(* CODESYS project XPlanarApplication206.library
   Version: 2.0.6
   Title: XPlanarApplication
   DefaultNamespace: XPlanarApplication
   Placeholder: XPlanarApplication
   Company: Beckhoff Automation LLC

Project tree, tasks and I/O mapping:
  libraries: Tc2_Math, * (Beckhoff Automation GmbH); Tc2_Standard, * (Beckhoff Automation GmbH); Tc2_System, * (Beckhoff Automation GmbH); Tc2_Utilities, * (Beckhoff Automation GmbH); Tc3_EventLogger, * (Beckhoff Automation GmbH); Tc3_Mc3PlanarMotion, * (Beckhoff Automation GmbH); Tc3_Module, * (Beckhoff Automation GmbH); Tc3_Physics, * (Beckhoff Automation GmbH); Tc3_XPlanarUtility, * (Beckhoff Automation GmbH)
  _Internal/
    HasPosition/
      function block FB_PositionXY [ST]: x, y
      interface I_HasPosition: x, y
    Interfaces/
      interface I_Base
      interface I_Cyclic: CyclicLogic
      interface I_Initializable: Initialize, Initialized
      interface I_Resettable: Reset
    Movers/
      ExernalAPI/
        DUT/
          data type ST_CommandResult
          data type ST_ExternalMoverCommand
          data type ST_ExternalMoverStatus
          data type ST_ExternalMoverTargetData
        function block FB_MoverExternalAPI [ST]: CyclicLogic, Disable, Enable, FB_Init, FreeMove, GetCurrentPosition, Halt, JoinClosestTrack, JoinTrack, LeaveTrack, Reset, Rotate, SendToStation, SquareUp, TiltA, TiltB, TrackMove, TrackMoveXY, VerticalMove
      MoverList/
        function block FB_MoverList [ST]: AddMover, Clear, Count, FirstMover, List, RemoveMover
        interface I_MoverList: AddMover, Clear, Count, FirstMover, List, RemoveMover
      MoverQueue/
        function block FB_MoverQueue [ST]: Clear, Count, Dequeue, Enqueue, FirstMover, Queue
        interface I_MoverQueue: Clear, Count, Dequeue, Enqueue, FirstMover, Queue
    NullObjects/
      function block FB_NullMover [ST]: ActualPosition, AddToGroup, AtRotationPosition, Busy, CommandLog, CyclicLogic, Destination, Disable, Dynamics, Enable, EnterMovementArea, Error, ErrorId, Gap, Halt, IdentifiedBTN, Initialize, InStation, LastCyclePosition, LeaveMovementArea, MoveCommand, MoverBTN, MoverData, MoverIndex, MoverType, pm, Reset, RotationModulo, Status, Utility
      function block FB_NullMoverData [ST]
      global variables NullObjects
    TaskBaseClasses/
      function block FB_MoverTask [ST]: CyclicLogic, FB_Init, UpdateLog
      function block FB_PartTask [ST]: Part
      function block FB_TaskResult [ST]: Aborted, BlockingObjectInfo, Busy, Done, Error, ErrorID, Result, TaskName
      function block FB_TrackTask [ST]: Track
      function block FB_XPlanarTaskBase [ST]: CyclicLogic, PlanarFeedback
      interface I_PlanarTaskResult: Aborted, BlockingObjectInfo, Busy, Done, Error, ErrorID
  Mover/
    DUTs/
      data type ST_CommandLog
      data type ST_MoveDynamics
      data type ST_MoverCommandInfo
      data type ST_MoverObjectInfos
    Interfaces/
      interface I_HasMoverData: MoverData
      interface I_MoveCommands: FreeMove, JoinClosestTrack, JoinTrack, LeaveTrack, MoveRelativeC, MoveRelativeX, MoveRelativeY, MoveVelocityX, MoveX, MoveY, Rotate, RunExternalSpAbsoluteMode, RunExternalSpRelativeMode, SendToStation, SquareUp, StopExternalSp, TiltA, TiltB, TrackMove, TrackMoveXY, VerticalMove
      interface I_MoveDynamics: Movement, Rotation, Tilt
      interface I_MoverData
      interface I_XPlanarMover: ActualPosition, AddToGroup, AtRotationPosition, Busy, CommandLog, CyclicLogic, Destination, Disable, Dynamics, Enable, EnterMovementArea, Error, ErrorId, Gap, Halt, IdentifiedBTN, Initialize, InStation, LastCyclePosition, LeaveMovementArea, MoveCommand, MoverBTN, MoverIndex, MoverType, pm, Reset, RotationModulo, Status, Utility
    TaskClasses/
      function block FB_AddToGroup [ST]: Execute
      function block FB_Disable [ST]: Execute
      function block FB_Enable [ST]: Execute
      function block FB_EnterMovementArea [ST]: CyclicLogic, Execute
      function block FB_Halt [ST]: Execute
      function block FB_JoinClosestTrack [ST]: CyclicLogic, Execute
      function block FB_JoinTrack [ST]: Execute
      function block FB_LeaveMovementArea [ST]: CyclicLogic, Execute
      function block FB_LeaveTrack [ST]: Execute
      function block FB_MoveA [ST]: Execute
      function block FB_MoveB [ST]: Execute
      function block FB_MoveRelativeC [ST]: Execute
      function block FB_MoveRelativeX [ST]: Execute
      function block FB_MoveRelativeY [ST]: Execute
      function block FB_MoveToPosition [ST]: Execute
      function block FB_MoveVelocityC [ST]: Execute
      function block FB_MoveVelocityX [ST]: Execute
      function block FB_MoveVelocityY [ST]: Execute
      function block FB_MoveX [ST]: Execute
      function block FB_MoveY [ST]: Execute
      function block FB_MoveZ [ST]: Execute
      function block FB_ResetMover [ST]: Execute
      function block FB_Rotate [ST]: Execute
      function block FB_RunExternalSetpointAbsoluteMode [ST]: Execute
      function block FB_RunExternalSetpointRelativeMode [ST]: Execute
      function block FB_SquareUp [ST]: CyclicLogic, Execute
      function block FB_StopExternalSetpoint [ST]: Execute
      function block FB_TrackMove [ST]: Execute
      function block FB_TrackMoveXY [ST]: Execute
    function block FB_XPlanarMover [ST]: Initialize, Initialized, FreeMove, JoinClosestTrack, JoinTrack, LeaveTrack, MoveRelativeC, MoveRelativeX, MoveRelativeY, MoveVelocityC, MoveVelocityX, MoveVelocityY, MoveX, MoveY, Rotate, RunExternalSpAbsoluteMode, RunExternalSpRelativeMode, SendToStation, SquareUp, StopExternalSp, TiltA, TiltB, TrackMove, TrackMoveXY, VerticalMove, Movement, Rotation, Tilt, ActualPosition, AddToGroup, AtRotationPosition, Busy, CommandLog, Destination, Disable, Dynamics, Enable, EnterMovementArea, Error, ErrorId, Gap, Halt, IdentifiedBTN, InStation, LeaveMovementArea, MoveCommand, MoverBTN, MoverIndex, MoverType, ObjectInfo, pm, Reset, RotationModulo, Status, Utility, CyclicLogic, FB_Init, LastCyclePosition, MoverData
  Part/
    Tasks/
      function block FB_AllowEnable [ST]: Execute
      function block FB_ForceDisable [ST]: Execute
      function block FB_Initialize [ST]: Execute
      function block FB_ResetPart [ST]: Execute
    function block FB_XPlanarPart [ST]: Busy, CyclicLogic, Error, ErrorId, ForceDisable, Initialize, ObjectID, pm, Reset, SetAllowEnable, State
    interface I_XPlanarPart: Busy, Error, ErrorId, ForceDisable, ObjectID, pm, Reset, SetAllowEnable, State
  PositionTrigger/
    function block FB_XPlanarPositionTrigger [ST]: CyclicLogic, DeregisterMover, GetMover, MoverIsPresent, MoverQueue, Position, RegisterAllMovers, RegisterMover, WatchForMover
    interface I_XPlanarPositionTrigger: DeregisterMover, GetMover, MoverIsPresent, MoverQueue, Position, RegisterAllMovers, RegisterMover
  Project Information/
    function F_GetCompany [ST]
    function F_GetTitle [ST]
    function F_GetVersion [ST]
  Station/
    DUT/
      data type E_StationType
      data type E_XplanarStationState
      data type ST_StationHMI
      data type ST_XPlanarStationObjectInfos
    Interfaces/
      interface I_HasProcess: Process
      interface I_StationProcess: Execute
    function block FB_XPlanarStationBase [ST]: Process, AllowQueing, CanReleaseMover, CurrentMover, Error, Execute, HasMover, ID, MoverList, NextStation, Position, Reset, Size, StationComplete, StationReady, StationType, TrackID, CyclicLogic, FB_Init, Name, WatchForMover
    interface I_XPlanarStation: AllowQueing, CanReleaseMover, CurrentMover, CyclicLogic, Execute, HasMover, ID, MoverList, Name, NextStation, Position, Reset, Size, StationComplete, StationReady, StationType, TrackID
  Tile/
    DUT/
      data type ST_TileObjectInfos
      data type ST_TileTemperatures
    function block FB_XPlanarTile [ST]: Btn, Busy, CyclicLogic, DcLinkOk, Error, ErrorId, Index, Initialize, PartIndex, PositionOnPart, Temperatures, TimeToShutdown, Update, Utility
    interface I_XPlanarTile: Btn, Busy, DcLinkOk, Error, ErrorId, Index, PartIndex, PositionOnPart, Temperatures, TimeToShutdown, Update, Utility
  Track/
    DUT/
      data type E_TrackItemType
      data type ST_TrackDefinition
      data type ST_TrackItems
      data type ST_TrackStatus
    TaskClasses/
      function block FB_AddTrackToGroup [ST]: Execute
      function block FB_AppendLine [ST]: Execute
      function block FB_AppendPoint [ST]: Execute
      function block FB_BuildTrack [ST]: CyclicLogic, Execute
      function block FB_ClearSegment [ST]: Execute
      function block FB_CloseLoop [ST]: Execute
      function block FB_DisableTrack [ST]: Execute
      function block FB_EnableTrack [ST]: Execute
      function block FB_SetEndAtTrack [ST]: Execute
      function block FB_SetStartFromTrack [ST]: Execute
      function block FB_TrackReset [ST]: Execute
    function block FB_XPlanarTrackSegment [ST]: Initialize, Initialized, AddToGroup, AppendLine, AppendPoint, Build, Busy, Clear, CloseLoop, Definition, Disable, Enable, Error, ErrorId, GetTrackPositionAt, Index, IsStanding, MoverCount, MovingMoverCount, pm, Reset, SetEndAtTrack, SetStartFromTrack, Status, TrackLength, Utility, CyclicLogic, FB_Init
    interface I_XPlanarTrack: AddToGroup, AppendLine, AppendPoint, Build, Busy, Clear, CloseLoop, CyclicLogic, Definition, Disable, Enable, Error, ErrorId, GetTrackPositionAt, Index, Initialize, MoverCount, MovingMoverCount, pm, Reset, Status, TrackLength, Utility
  Version/
    global variables Global_Version
  XPlanarComponent/
    TaskClasses/
      function block FB_AbortSystem [ST]: CyclicLogic, Execute
      function block FB_EnableGroup [ST]: Execute
      function block FB_MoverIdentification [ST]: CyclicLogic, Execute
      function block FB_MoverRedetection [ST]: CyclicLogic, Execute, MoverDetectionInfo
      function block FB_ResetGroup [ST]: Execute
      function block FB_ResetXPlanar [ST]: CyclicLogic, Execute
    function block FB_Component_XPlanar [ST]: CyclicLogic, Initialize, Initialized, Abort, AddMoversToGroup, AddTracksToGroup, DisableMovers, EnableGroup, EnableMovers, EnableTracks, Halt, IdentifyMovers, Monitoring, MoverDetectionInfo, MoverRedetect, Reset, Utility
    interface I_XPlanarSystem: Abort, AddMoversToGroup, AddTracksToGroup, DisableMovers, EnableGroup, EnableMovers, EnableTracks, Halt, IdentifyMovers, MoverDetectionInfo, MoverRedetect, Reset, Utility
  global variables HMIObjectCounts
  global variables ip
  00000000-0000-0000-0000-000000000000|LICENSE
  LICENSE
  global variables SystemParameters
  global variables XPlanar
  global variables XPlanarHMI
*)

// _Internal/Movers/ExernalAPI/DUT/ST_CommandResult
TYPE ST_CommandResult :
STRUCT
	Busy	: BOOL;
	Done	: BOOL;
	Aborted	: BOOL;
	Error	: BOOL;
	ErrorId	: UDINT;
END_STRUCT
END_TYPE

// _Internal/Movers/ExernalAPI/DUT/ST_ExternalMoverCommand
TYPE ST_ExternalMoverCommand :
	STRUCT
		Enable		 : BOOL;
		Disable		 : BOOL;
		Reset		 : BOOL;
		Halt		 : BOOL;
		FreeMove	 : BOOL;
		Rotate		 : BOOL;
		TiltA		 : BOOL;
		TiltB		 : BOOL;
		VerticalMove : BOOL;
		TrackMove	 : BOOL;
		TrackMoveXY	 : BOOL;
		JoinTrack	 : BOOL;
		LeaveTrack	 : BOOL;
		SquareUp	 : BOOL;
	END_STRUCT
END_TYPE

// _Internal/Movers/ExernalAPI/DUT/ST_ExternalMoverStatus
TYPE ST_ExternalMoverStatus :
	STRUCT
		Enabled		   : BOOL;
		Error		   : BOOL;
		InStation	   : BOOL;
		ErrorID		   : UDINT;
		CurrentStation : STRING;
		CommandMode	   : STRING;
		LastCommand	   : STRING;
	END_STRUCT
END_TYPE

// _Internal/Movers/ExernalAPI/DUT/ST_ExternalMoverTargetData
TYPE ST_ExternalMoverTargetData :
	STRUCT
		Position	: Tc3_Mc3PlanarMotion.MoverVector;
		TargetStationID : UDINT;
		TargetTrackID	: UDINT;
		TrackPosition	: LREAL;
		TrackDirection	: UINT;
		TrackGap		: LREAL;
	END_STRUCT
END_TYPE

// Mover/DUTs/ST_CommandLog
TYPE ST_CommandLog EXTENDS ST_MoverCommandInfo :
	STRUCT
		Timestamp : STRING(24);
	END_STRUCT
END_TYPE

// Mover/DUTs/ST_MoveDynamics
TYPE ST_MoveDynamics :
STRUCT
	Velocity	: LREAL;
	Accel		: LREAL;
	Decel		: LREAL;
	Jerk		: LREAL;
END_STRUCT
END_TYPE

// Mover/DUTs/ST_MoverCommandInfo
TYPE ST_MoverCommandInfo :
	STRUCT
		Command	 : STRING;
		Velocity : LREAL;
		Accel	 : LREAL;
		Decel	 : LREAL;
		Jerk	 : LREAL;
	END_STRUCT
END_TYPE

// Mover/DUTs/ST_MoverObjectInfos
TYPE ST_MoverObjectInfos :
	STRUCT
		Width	 : DINT;
		Height	 : DINT;
		MoverBTN : STRING(13);
		Error	 : BOOL;
	END_STRUCT
END_TYPE

// Station/DUT/E_StationType
{attribute 'qualified_only'}
TYPE E_StationType : (
		Process		  := 0,
		DecisionPoint := 1,
		MultiMover	  := 2
	) UDINT;
END_TYPE

// Station/DUT/E_XplanarStationState
{attribute 'qualified_only'}
{attribute 'strict'}
{attribute 'to_string'}
TYPE E_XplanarStationState : (
		StationIdle := 0,
		ProcessMover,
		SquareUpMover,
		SendMoverAway,
		CycleComplete,
		SendQueue,
		StationError
	);
END_TYPE

// Station/DUT/ST_StationHMI
TYPE ST_StationHMI :
	STRUCT
		Error		   : BOOL;
		Reset		   : BOOL;
		StationReady   : BOOL;
		HasMover	   : BOOL;
		CurrentMoverID : STRING(13);
		CurrentState   : STRING;
	END_STRUCT
END_TYPE

// Station/DUT/ST_XPlanarStationObjectInfos
TYPE ST_XPlanarStationObjectInfos :
	STRUCT
		X	   : DINT;
		Y	   : DINT;
		Width  : DINT;
		Height : DINT;
	END_STRUCT
END_TYPE

// Tile/DUT/ST_TileObjectInfos
TYPE ST_TileObjectInfos :
	STRUCT
		X	   : DINT;
		Y	   : DINT;
		Width  : DINT;
		Height : DINT;
	END_STRUCT
END_TYPE

// Tile/DUT/ST_TileTemperatures
TYPE ST_TileTemperatures :
	STRUCT
		Center : LREAL;
		East   : LREAL;
		West   : LREAL;
		North  : LREAL;
		South  : LREAL;
	END_STRUCT
END_TYPE

// Track/DUT/E_TrackItemType
TYPE E_TrackItemType :
(
	Point := 0,
	Line,
	Circle
);
END_TYPE

// Track/DUT/ST_TrackDefinition
TYPE ST_TrackDefinition :
	STRUCT
		StartFromTrackID : UDINT;
		EndAtTrackID	 : UDINT;
		CloseLoop		 : BOOL;
		Items			 : ARRAY[1..SystemParameters.MAX_OBJECTS_PER_TRACK] OF ST_TrackItems;
	END_STRUCT
END_TYPE

// Track/DUT/ST_TrackItems
TYPE ST_TrackItems :
STRUCT
	ItemType		: E_TrackItemType;
	StartPoint		: PositionXYC;
	EndPoint		: PositionXYC;
	CenterPoint		: PositionXY;
	CircleClockwise : BOOL;
END_STRUCT
END_TYPE

// Track/DUT/ST_TrackStatus
TYPE ST_TrackStatus :
	STRUCT
		State			 : MC_PLANAR_STATE;
		OperationMode	 : MC_PLANAR_TRACK_OPERATION_MODE;
		MoverCount		 : UDINT;
		CalculatedLength : LREAL;
	END_STRUCT
END_TYPE

// _Internal/NullObjects/NullObjects
{attribute 'qualified_only'}
VAR_GLOBAL
	MoverData	 : FB_NullMoverData;
	XPlanarMover : FB_NullMover;
END_VAR

// Version/Global_Version
{attribute 'TcGenerated'}
{attribute 'no-analysis'}
{attribute 'linkalways'}
// This function has been automatically generated from the project information.
VAR_GLOBAL CONSTANT
	{attribute 'const_non_replaced'}
	stLibVersion_XPlanarApplication : ST_LibVersion := (iMajor := 2, iMinor := 0, iBuild := 6, iRevision := 0, nFlags := 0, sVersion := '2.0.6');
END_VAR

// HMIObjectCounts
{attribute 'qualified_only'}
VAR_GLOBAL CONSTANT
	Movers	 : UINT := 10; //Total number of movers configured in the system
	Tiles	 : UINT := 10; //Total number of track segments in the system
	Stations : UINT := 10; //Total number of stations for HMI array size
END_VAR

// ip
{attribute 'qualified_only'}
VAR_GLOBAL
	Movers	 : ARRAY[0..Param_TcIoXPlanarEnvironment.MaxMcPlanarMovers] OF I_XPlanarMover;
	Tracks	 : ARRAY[0..Param_TcIoXPlanarEnvironment.MaxTracks] OF I_XPlanarTrack;
	Stations : ARRAY[0..SystemParameters.MAX_STATION_COUNT] OF I_XPlanarStation;
END_VAR

// SystemParameters
{attribute 'qualified_only'}
VAR_GLOBAL CONSTANT
	MAX_LOG_COUNT	 	  : UINT  := 20; //Size of command mover log
	MAX_OBJECTS_PER_TRACK : UINT  := 20;  //Maximum number of points or lines defined in a single track segment
	MAX_STATION_COUNT	  : UINT  := 100; //Total number of stations in the system
	FastEnable			  : BOOL := TRUE;
	AutoDynamicsReduction : BOOL := TRUE;
END_VAR

// XPlanar
{attribute 'qualified_only'}
VAR_GLOBAL
	Environment		   : Tc3_MC3PlanarMotion.MC_PlanarEnvironment; //This gets linked to the Environment object in the XPlanar MC Project
	EnvironmentTcIo	   : Tc3_XPlanarUtility.FB_TcIoXPlanarEnvironment; //This profides an interface to the XPlanar TcCom objects
	Group			   : Tc3_MC3PlanarMotion.MC_PlanarGroup;
	Parts			   : ARRAY[1..Param_TcIoXPlanarEnvironment.MaxParts] OF FB_XPlanarPart;
	Tiles			   : ARRAY[1..Param_TcIoXPlanarEnvironment.MaxTiles] OF FB_XPlanarTile;
	OperationMode	   : XPlanarOperationMode;
	RotationMultiplier : LREAL := 120.0;
	XPUCount		   : UINT;
	PartCount		   : UINT;
	TrackCount		   : UDINT;
	MoverCount		   : UDINT;
	StationCount	   : UDINT;
	TileCount		   : UINT;
END_VAR

// XPlanarHMI
{attribute 'qualified_only'}
VAR_GLOBAL
	{ attribute 'TcHmiSymbol.AddSymbol' }
	{ attribute 'TcHmiSymbol.AddSymbol.UserGroups' := '__SystemAdministrators,Admin'}
	MoverObjects : ARRAY[1..Tc3_XPlanarUtility.Param_TcIoXPlanarEnvironment.MaxXPlanarMoversPerXpu] OF ST_MoverObjectInfos;
	{ attribute 'TcHmiSymbol.AddSymbol' }
	{ attribute 'TcHmiSymbol.AddSymbol.UserGroups' := '__SystemAdministrators,Admin'}
	MoverPositions : ARRAY[1..Tc3_XPlanarUtility.Param_TcIoXPlanarEnvironment.MaxXPlanarMoversPerXpu] OF MoverVector;
	{ attribute 'TcHmiSymbol.AddSymbol' }
	{ attribute 'TcHmiSymbol.AddSymbol.UserGroups' := '__SystemAdministrators,Admin'}
	TileObjects : ARRAY[1..Tc3_XPlanarUtility.Param_TcIoXPlanarEnvironment.MaxTiles] OF ST_TileObjectInfos;
	{ attribute 'TcHmiSymbol.AddSymbol' }
	{ attribute 'TcHmiSymbol.AddSymbol.UserGroups' := '__SystemAdministrators,Admin'}
	StationObjects : ARRAY[1..SystemParameters.MAX_STATION_COUNT] OF ST_XPlanarStationObjectInfos;
END_VAR

// _Internal/HasPosition/FB_PositionXY
FUNCTION_BLOCK FB_PositionXY IMPLEMENTS I_HasPosition
VAR
	_x	: LREAL;
	_y	: LREAL;
END_VAR

PROPERTY x : LREAL
GET
x := _x;
END_GET
SET
_x := x;
END_SET
END_PROPERTY

PROPERTY y : LREAL
GET
y := _y;
END_GET
SET
_y := y;
END_SET
END_PROPERTY

END_FUNCTION_BLOCK

// _Internal/HasPosition/I_HasPosition
INTERFACE I_HasPosition EXTENDS I_Base

PROPERTY x : LREAL
GET
END_GET
SET
END_SET
END_PROPERTY

PROPERTY y : LREAL
GET
END_GET
SET
END_SET
END_PROPERTY

END_INTERFACE

// _Internal/Interfaces/I_Base
INTERFACE I_Base EXTENDS __System.IQueryInterface

END_INTERFACE

// _Internal/Interfaces/I_Cyclic
INTERFACE I_Cyclic EXTENDS I_Base

METHOD CyclicLogic
END_METHOD

END_INTERFACE

// _Internal/Interfaces/I_Initializable
INTERFACE I_Initializable EXTENDS I_Base

METHOD Initialize
END_METHOD

{attribute 'monitoring' := 'call'}
PROPERTY Initialized : BOOL
GET
END_GET
SET
END_SET
END_PROPERTY

END_INTERFACE

// _Internal/Interfaces/I_Resettable
INTERFACE I_Resettable EXTENDS I_Base

METHOD Reset
END_METHOD

END_INTERFACE

// _Internal/Movers/ExernalAPI/FB_MoverExternalAPI
FUNCTION_BLOCK FB_MoverExternalAPI IMPLEMENTS I_Cyclic
VAR
	_Mover				  : I_XPlanarMover;
	ipCommandResult		  : I_PlanarTaskResult;
	
	//Input Data
	MoverCommands  AT %I* : ST_ExternalMoverCommand;
	TargetData	   AT %I* : ST_ExternalMoverTargetData;
	MoveDynamics   AT %I* : ST_MoveDynamics;
	RotateDynamics AT %I* : ST_MoveDynamics;
	TiltDynamics   AT %I* : ST_MoveDynamics;
	
	//Output Data
	CommandResult  AT %Q* : ST_CommandResult;
	MoverStatus	   AT %Q* : ST_ExternalMoverStatus;
END_VAR

METHOD CyclicLogic
VAR_INST
	TargetModulo : LREAL;
	TargetTurns	 : DINT;
END_VAR
IF ipCommandResult <> 0 THEN
	CommandResult.Busy	  := ipCommandResult.Busy;
	CommandResult.Done	  := ipCommandResult.Done;
	CommandResult.Error	  := ipCommandResult.Error;
	CommandResult.ErrorID := ipCommandResult.ErrorID;
	CommandResult.Aborted := ipCommandResult.Aborted;
END_IF

IF _Mover <> 0 THEN
	IF MoverCommands.Enable THEN
		Enable();
	END_IF

	IF MoverCommands.Disable THEN
		Disable();
	END_IF

	IF MoverCommands.Reset THEN
		Reset();
	END_IF

	IF MoverCommands.Halt THEN
		Halt();
	END_IF

	IF MoverCommands.FreeMove THEN
		FreeMove(X := TargetData.Position.x, Y := TargetData.Position.y);
	END_IF

	IF MoverCommands.Rotate THEN
		IF TargetData.Position.c > 360 THEN
			TargetModulo := LMOD(TargetData.Position.c, 360);
			TargetTurns	 := MODTURNS(TargetData.Position.c, 360);
		ELSE
			TargetModulo := TargetData.Position.c;
			TargetTurns	 := 0;
		END_IF

		Rotate(TargetModulo, TargetTurns);
	END_IF
	
	IF MoverCommands.TiltA THEN
		TiltA(TargetData.Position.a);
	END_IF
	
	IF MoverCommands.TiltB THEN
		TiltB(TargetData.Position.b);
	END_IF
	
	IF MoverCommands.VerticalMove THEN
		VerticalMove(TargetData.Position.z);
	END_IF	
	
	IF MoverCommands.TrackMove THEN
		TrackMove(TargetData.TargetTrackID, TargetData.TrackPosition, TargetData.TrackGap, TargetData.TrackDirection);
	END_IF
	
	IF MoverCommands.TrackMoveXY THEN
		TrackMoveXY(X := TargetData.Position.x, TargetData.Position.y, TargetData.TrackGap, TargetData.TargetTrackID, TargetData.TrackDirection);
	END_IF	
	
	IF MoverCommands.JoinTrack THEN
		JoinTrack(TargetData.TargetTrackID);
	END_IF
	
	IF MoverCommands.LeaveTrack THEN
		LeaveTrack(TargetData.Position.x, TargetData.Position.y);
	END_IF
END_IF
END_METHOD

{attribute 'TcRpcEnable'}
METHOD Disable : BOOL
ipCommandResult := _Mover.Disable();
Disable := TRUE;
END_METHOD

{attribute 'TcRpcEnable'}
METHOD Enable : BOOL
ipCommandResult := _Mover.Enable();
Enable := TRUE;
END_METHOD

//FB_Init is always available implicitly and it is used primarily for initialization.
//The return value is not evaluated. For a specific influence, you can also declare the
//methods explicitly and provide additional code there with the standard initialization
//code. You can evaluate the return value.
METHOD FB_Init : BOOL
VAR_INPUT
	bInitRetains : BOOL; // TRUE: the retain variables are initialized (reset warm / reset cold)
	bInCopyCode	 : BOOL; // TRUE: the instance will be copied to the copy code afterward (online change)   
	Mover		 : I_XPlanarMover;
END_VAR
_Mover := Mover;
END_METHOD

{attribute 'TcRpcEnable'}
METHOD FreeMove : BOOL
VAR_INPUT
	X		: LREAL;
	Y		: LREAL;
END_VAR
IF X > 0 AND Y > 0 THEN
	ipCommandResult := _Mover.MoveCommand.FreeMove(X, Y);
	FreeMove := TRUE;
END_IF
END_METHOD

{attribute 'TcRpcEnable'}
METHOD GetCurrentPosition : Tc3_Mc3PlanarMotion.MoverVector
GetCurrentPosition := _Mover.ActualPosition;
END_METHOD

{attribute 'TcRpcEnable'}
METHOD Halt : BOOL
ipCommandResult := _Mover.Halt();
Halt := TRUE;
END_METHOD

{attribute 'TcRpcEnable'}
METHOD JoinClosestTrack : BOOL
ipCommandResult := _Mover.MoveCommand.JoinClosestTrack();
JoinClosestTrack := TRUE;
END_METHOD

{attribute 'TcRpcEnable'}
METHOD JoinTrack : BOOL
VAR_INPUT
	TrackId		: UDINT;
END_VAR
IF TrackId > 0 AND TrackID <= XPlanar.TrackCount THEN
	ipCommandResult := _Mover.MoveCommand.JoinTrack(ip.Tracks[TrackId]);
	JoinTrack := TRUE;
END_IF
END_METHOD

{attribute 'TcRpcEnable'}
METHOD LeaveTrack : BOOL
VAR_INPUT
	X   : LREAL;
	Y   : LREAL;
END_VAR
IF X > 0 AND Y > 0 THEN
	ipCommandResult := _Mover.MoveCommand.LeaveTrack(X, Y);
	LeaveTrack := TRUE;
END_IF
END_METHOD

{attribute 'TcRpcEnable'}
METHOD Reset : BOOL
ipCommandResult := _Mover.Reset();
Reset := TRUE;
END_METHOD

METHOD Rotate : BOOL
VAR_INPUT
	Position		: LREAL;
	AdditionalTurns : DINT := 0;
END_VAR
ipCommandResult := _Mover.MoveCommand.Rotate(Position, AdditionalTurns);
Rotate := TRUE;
END_METHOD

{attribute 'TcRpcEnable'}
METHOD SendToStation : BOOL
VAR_INPUT
	StationId		: UDINT;
END_VAR
IF StationId > 0 AND StationId <= XPlanar.StationCount THEN
	ipCommandResult := _Mover.MoveCommand.SendToStation(ip.Stations[StationId]);
	SendToStation := TRUE;
END_IF
END_METHOD

{attribute 'TcRpcEnable'}
METHOD SquareUp : BOOL
ipCommandResult := _Mover.MoveCommand.SquareUp();
SquareUp := TRUE;
END_METHOD

{attribute 'TcRpcEnable'}
METHOD TiltA : BOOL
VAR_INPUT
	Position	: LREAL;
END_VAR
ipCommandResult := _Mover.MoveCommand.TiltA(Position);
TiltA := TRUE;
END_METHOD

{attribute 'TcRpcEnable'}
METHOD TiltB : BOOL
VAR_INPUT
	Position	: LREAL;
END_VAR
ipCommandResult := _Mover.MoveCommand.TiltB(Position);
TiltB := TRUE;
END_METHOD

{attribute 'TcRpcEnable'}
METHOD TrackMove : BOOL
VAR_INPUT
	TrackId		: UDINT;
	Position	: LREAL;
	Gap			: LREAL;
	Direction	: UINT;
END_VAR
IF TrackId > 0 AND TrackId <= XPlanar.TrackCount THEN
	ipCommandResult := _Mover.MoveCommand.TrackMove(Position, Gap, ip.Tracks[TrackId], Direction);
	TrackMove := TRUE;
END_IF
END_METHOD

{attribute 'TcRpcEnable'}
METHOD TrackMoveXY : BOOL
VAR_INPUT
	X		  : LREAL;
	Y		  : LREAL;
	Gap		  : LREAL;
	TrackId	  : UDINT;
	Direction : UINT := 1;
END_VAR
IF TrackId > 0 AND TrackId <= XPlanar.TrackCount THEN
	ipCommandResult := _Mover.MoveCommand.TrackMoveXY(X, Y, Gap, ip.Tracks[TrackId], Direction);
	TrackMoveXY := TRUE;
END_IF
END_METHOD

{attribute 'TcRpcEnable'}
METHOD VerticalMove : BOOL
VAR_INPUT
	Position	: LREAL;
END_VAR
ipCommandResult := _Mover.MoveCommand.VerticalMove(Position);
VerticalMove := TRUE;
END_METHOD

END_FUNCTION_BLOCK

// Mover/Interfaces/I_XPlanarMover
INTERFACE I_XPlanarMover EXTENDS I_Base, I_HasMoverData

{attribute 'suppress_wrn_C0410'}
PROPERTY ActualPosition : REFERENCE TO MoverVector
GET
END_GET
END_PROPERTY

METHOD AddToGroup : I_PlanarTaskResult
VAR_INPUT
	PlanarGroup : REFERENCE TO MC_PlanarGroup;
END_VAR
END_METHOD

PROPERTY AtRotationPosition : BOOL
GET
END_GET
END_PROPERTY

PROPERTY Busy : BOOL
GET
END_GET
END_PROPERTY

{attribute 'suppress_wrn_C0410'}
PROPERTY CommandLog : REFERENCE TO ARRAY [0..SystemParameters.MAX_LOG_COUNT] of ST_CommandLog
GET
END_GET
END_PROPERTY

METHOD CyclicLogic
END_METHOD

PROPERTY Destination : I_XPlanarStation
GET
END_GET
SET
END_SET
END_PROPERTY

METHOD Disable : I_PlanarTaskResult
END_METHOD

PROPERTY Dynamics : I_MoveDynamics
GET
END_GET
END_PROPERTY

METHOD Enable : I_PlanarTaskResult
END_METHOD

METHOD EnterMovementArea : I_PlanarTaskResult
VAR_INPUT
	PartId		: OTCID;
	PositionX	: LREAL;
	PositionY	: LREAL;
END_VAR
END_METHOD

PROPERTY Error : BOOL
GET
END_GET
END_PROPERTY

PROPERTY ErrorId : UDINT
GET
END_GET
END_PROPERTY

PROPERTY Gap : LREAL
GET
END_GET
SET
END_SET
END_PROPERTY

METHOD Halt : I_PlanarTaskResult
END_METHOD

PROPERTY IdentifiedBTN : STRING
GET
END_GET
SET
END_SET
END_PROPERTY

{attribute 'hide'}
METHOD Initialize
END_METHOD

PROPERTY InStation : BOOL
GET
END_GET
SET
END_SET
END_PROPERTY

PROPERTY LastCyclePosition : Reference TO MoverVector
GET
END_GET
END_PROPERTY

METHOD LeaveMovementArea : I_PlanarTaskResult
END_METHOD

PROPERTY MoveCommand : I_MoveCommands
GET
END_GET
END_PROPERTY

PROPERTY MoverBTN : STRING
GET
END_GET
END_PROPERTY

PROPERTY MoverIndex : UDINT
GET
END_GET
SET
END_SET
END_PROPERTY

PROPERTY MoverType : XplanarMoverType
GET
END_GET
SET
END_SET
END_PROPERTY

{attribute 'suppress_wrn_C0410'}
PROPERTY pm : REFERENCE TO MC_PlanarMover
GET
END_GET
END_PROPERTY

METHOD PUBLIC Reset : I_PlanarTaskResult
END_METHOD

PROPERTY RotationModulo : LREAL
GET
END_GET
END_PROPERTY

{attribute 'suppress_wrn_C0410'}
PROPERTY Status : REFERENCE TO CDT_MCTOPLC_PLANAR_MOVER_STD
GET
END_GET
END_PROPERTY

PROPERTY Utility : I_TcIoXPlanarMover
GET
END_GET
SET
END_SET
END_PROPERTY

END_INTERFACE

// Mover/Interfaces/I_HasMoverData
INTERFACE I_HasMoverData EXTENDS I_Base

PROPERTY MoverData : I_MoverData
GET
END_GET
SET
END_SET
END_PROPERTY

END_INTERFACE

// Mover/Interfaces/I_MoverData
INTERFACE I_MoverData EXTENDS I_Base

END_INTERFACE

// _Internal/TaskBaseClasses/I_PlanarTaskResult
INTERFACE I_PlanarTaskResult

{attribute 'monitoring' := 'call'}
PROPERTY Aborted : BOOL
GET
END_GET
END_PROPERTY

{attribute 'suppress_wrn_C0410'}
PROPERTY BlockingObjectInfo : REFERENCE TO PlanarObjectInfo
GET
END_GET
END_PROPERTY

{attribute 'monitoring' := 'call'}
PROPERTY Busy : BOOL
GET
END_GET
END_PROPERTY

{attribute 'monitoring' := 'call'}
PROPERTY Done : BOOL
GET
END_GET
END_PROPERTY

{attribute 'monitoring' := 'call'}
PROPERTY Error : BOOL
GET
END_GET
END_PROPERTY

{attribute 'monitoring' := 'call'}
PROPERTY ErrorID : UDINT
GET
END_GET
END_PROPERTY

END_INTERFACE

// Station/I_XPlanarStation
INTERFACE I_XPlanarStation EXTENDS I_Base, I_HasProcess

PROPERTY AllowQueing : BOOL
GET
END_GET
SET
END_SET
END_PROPERTY

PROPERTY CanReleaseMover : BOOL
SET
END_SET
END_PROPERTY

PROPERTY CurrentMover : I_XPlanarMover
GET
END_GET
END_PROPERTY

{attribute 'hide'}
METHOD CyclicLogic
END_METHOD

METHOD Execute
END_METHOD

PROPERTY HasMover : BOOL
GET
END_GET
SET
END_SET
END_PROPERTY

PROPERTY ID : UDINT
GET
END_GET
SET
END_SET
END_PROPERTY

{attribute 'suppress_wrn_C0410'}
PROPERTY MoverList : REFERENCE TO FB_MoverList
GET
END_GET
END_PROPERTY

PROPERTY Name : STRING
GET
END_GET
SET
END_SET
END_PROPERTY

PROPERTY NextStation : I_XPlanarStation
GET
END_GET
SET
END_SET
END_PROPERTY

{attribute 'suppress_wrn_C0410'}
PROPERTY Position : REFERENCE TO PositionXYC
GET
END_GET
END_PROPERTY

METHOD Reset : BOOL
END_METHOD

{attribute 'suppress_wrn_C0410'}
PROPERTY Size : REFERENCE TO Position2D_LREAL
GET
END_GET
END_PROPERTY

PROPERTY StationComplete : BOOL
SET
END_SET
END_PROPERTY

PROPERTY StationReady : BOOL
GET
END_GET
END_PROPERTY

PROPERTY StationType : E_StationType
GET
END_GET
SET
END_SET
END_PROPERTY

PROPERTY TrackID : UDINT
GET
END_GET
SET
END_SET
END_PROPERTY

END_INTERFACE

// Station/Interfaces/I_HasProcess
INTERFACE I_HasProcess EXTENDS I_Base

PROPERTY Process : I_StationProcess
GET
END_GET
SET
END_SET
END_PROPERTY

END_INTERFACE

// Station/Interfaces/I_StationProcess
INTERFACE I_StationProcess EXTENDS I_Base

METHOD Execute : BOOL
VAR_INPUT
	Mover : I_XPlanarMover;
END_VAR
END_METHOD

END_INTERFACE

// _Internal/Movers/MoverList/FB_MoverList
FUNCTION_BLOCK FB_MoverList IMPLEMENTS I_MoverList
VAR
	MoversInList : UDINT := 0;
	ipMovers	  : ARRAY[1..Tc3_XPlanarUtility.Param_TcIoXPlanarEnvironment.MaxMcPlanarMovers] OF I_XPlanarMover;
END_VAR

METHOD AddMover : BOOL
VAR_INPUT
	ipMover : I_XPlanarMover;
END_VAR
IF MoversInList < Tc3_XPlanarUtility.Param_TcIoXPlanarEnvironment.MaxMcPlanarMovers THEN
	MoversInList			:= MoversInList + 1;
	ipMovers[MoversInList] := ipMover;
	AddMover					:= TRUE;
END_IF
END_METHOD

//=============================================================================
//	Method Clear()
//=============================================================================
//
//	Brute force reset of buffer
//
//-----------------------------------------------------------------------------
METHOD Clear : BOOL
MEMSET(ADR(ipMovers), 0, SIZEOF(ipMovers));
MoversInList := 0;
Clear		  := TRUE;
END_METHOD

PROPERTY Count : UDINT
GET
VAR
	i	 : UDINT;
	temp : UDINT;
END_VAR
Count := MoversInList;
END_GET
END_PROPERTY

PROPERTY FirstMover : I_XPlanarMover
GET
IF MoversInList > 0 THEN
	FirstMover := ipMovers[1];
END_IF
END_GET
END_PROPERTY

{attribute 'suppress_wrn_C0410'}
PROPERTY List : REFERENCE TO ARRAY[1..Tc3_XPlanarUtility.Param_TcIoXPlanarEnvironment.MaxMcPlanarMovers] OF I_XPlanarMover;
GET
VAR
	i : UDINT;
END_VAR
List ref= ipMovers;
END_GET
END_PROPERTY

METHOD RemoveMover
VAR_INPUT
	Mover	: I_XPlanarMover;
END_VAR
VAR
	i	: UDINT;
END_VAR
FOR i := 1 TO MoversInList DO
	IF ipMovers[i] = Mover THEN
		ipMovers[i] := 0;
	END_IF
END_FOR
//Todo: Repack the list
END_METHOD

END_FUNCTION_BLOCK

// _Internal/Movers/MoverList/I_MoverList
INTERFACE I_MoverList EXTENDS I_Base

METHOD AddMover : BOOL
VAR_INPUT
	ipMover : I_XPlanarMover;
END_VAR
END_METHOD

//=============================================================================
//	Method Clear()
//=============================================================================
//
//	Brute force reset of buffer
//
//-----------------------------------------------------------------------------
METHOD Clear : BOOL
END_METHOD

PROPERTY Count : UDINT
GET
END_GET
END_PROPERTY

PROPERTY FirstMover : I_XPlanarMover
GET
END_GET
END_PROPERTY

{attribute 'suppress_wrn_C0410'}
PROPERTY List : REFERENCE TO ARRAY[1..Tc3_XPlanarUtility.Param_TcIoXPlanarEnvironment.MaxMcPlanarMovers] OF I_XPlanarMover;
GET
END_GET
END_PROPERTY

METHOD RemoveMover
VAR_INPUT
	Mover	: I_XPlanarMover;
END_VAR
END_METHOD

END_INTERFACE

// Mover/Interfaces/I_MoveDynamics
INTERFACE I_MoveDynamics EXTENDS __SYSTEM.IQueryInterface

{attribute 'suppress_wrn_C0410'}
PROPERTY Movement : REFERENCE TO ST_MoveDynamics
GET
END_GET
END_PROPERTY

{attribute 'suppress_wrn_C0410'}
PROPERTY Rotation : REFERENCE TO ST_MoveDynamics
GET
END_GET
END_PROPERTY

{attribute 'suppress_wrn_C0410'}
PROPERTY Tilt : REFERENCE TO ST_MoveDynamics
GET
END_GET
END_PROPERTY

END_INTERFACE

// Mover/Interfaces/I_MoveCommands
INTERFACE I_MoveCommands EXTENDS __SYSTEM.IQueryInterface

METHOD FreeMove : I_PlanarTaskResult
VAR_INPUT
	XTarget			: LREAL;
	YTarget			: LREAL;
	CTarget			: LREAL := 0;
	Rototranslation : BOOL	:= FALSE;
END_VAR
END_METHOD

METHOD JoinClosestTrack : I_PlanarTaskResult
VAR_INPUT
	UseOrientation : BOOL := FALSE;
END_VAR
END_METHOD

METHOD JoinTrack : I_PlanarTaskResult
VAR_INPUT
	ipTrack		   : I_XPlanarTrack;
	UseOrientation : BOOL := FALSE;
END_VAR
END_METHOD

METHOD LeaveTrack : I_PlanarTaskResult
VAR_INPUT
	DestinationX   : LREAL;
	DestinationY   : LREAL;
	UseOrientation : BOOL := FALSE;
END_VAR
END_METHOD

METHOD MoveRelativeC : I_PlanarTaskResult
VAR_INPUT
	Distance	: LREAL;
END_VAR
END_METHOD

METHOD MoveRelativeX : I_PlanarTaskResult
VAR_INPUT
	Distance	: LREAL;
END_VAR
END_METHOD

METHOD MoveRelativeY : I_PlanarTaskResult
VAR_INPUT
	Distance	: LREAL;
END_VAR
END_METHOD

METHOD MoveVelocityX : I_PlanarTaskResult
VAR_INPUT
	Velocity	: LREAL;
END_VAR
END_METHOD

METHOD MoveX : I_PlanarTaskResult
VAR_INPUT
	Position	: LREAL;
END_VAR
END_METHOD

METHOD MoveY : I_PlanarTaskResult
VAR_INPUT
	Position	: LREAL;
END_VAR
END_METHOD

METHOD Rotate : I_PlanarTaskResult
VAR_INPUT
	Position		: LREAL;
	AdditionalTurns : DINT := 0;
END_VAR
END_METHOD

METHOD RunExternalSpAbsoluteMode : I_PlanarTaskResult
VAR_INPUT
	Position	 : MoverVector;
	Velocity	 : MoverVector;
	Acceleration : MoverVector;
END_VAR
END_METHOD

METHOD RunExternalSpRelativeMode : I_PlanarTaskResult
VAR_INPUT
	Position	 : MoverVector;
	Velocity	 : MoverVector;
	Acceleration : MoverVector;
END_VAR
END_METHOD

METHOD SendToStation : I_PlanarTaskResult
VAR_INPUT
	Destination : I_XPlanarStation;
END_VAR
END_METHOD

METHOD SquareUp : I_PlanarTaskResult
END_METHOD

METHOD StopExternalSp : I_PlanarTaskResult
END_METHOD

METHOD TiltA : I_PlanarTaskResult
VAR_INPUT
	Position : LREAL;
END_VAR
END_METHOD

METHOD TiltB : I_PlanarTaskResult
VAR_INPUT
	Position : LREAL;
END_VAR
END_METHOD

METHOD TrackMove : I_PlanarTaskResult
VAR_INPUT
	Position  : LREAL;
	Gap		  : LREAL;
	Track	  : I_XPlanarTrack;
	Direction : Tc3_Mc3PlanarMotion.MC_DIRECTION;
END_VAR
END_METHOD

METHOD TrackMoveXY : I_PlanarTaskResult
VAR_INPUT
	XPosition : LREAL;
	YPosition : LREAL;
	Gap		  : LREAL;
	Track	  : I_XPlanarTrack;
	Direction : Tc3_Mc3PlanarMotion.MC_DIRECTION;
END_VAR
END_METHOD

METHOD VerticalMove : I_PlanarTaskResult
VAR_INPUT
	Position : LREAL;
END_VAR
END_METHOD

END_INTERFACE

// Track/I_XPlanarTrack
INTERFACE I_XPlanarTrack EXTENDS __SYSTEM.IQueryInterface

METHOD AddToGroup : I_PlanarTaskResult
VAR_INPUT
	PlanarGroup : REFERENCE TO MC_PlanarGroup;
END_VAR
END_METHOD

METHOD AppendLine : I_PlanarTaskResult
VAR_INPUT
	StartPointX : LREAL;
	StartPointY : LREAL;
	EndPointX	: LREAL;
	EndPointY	: LREAL;
END_VAR
END_METHOD

METHOD AppendPoint : I_PlanarTaskResult
VAR_INPUT
	XPoint : LREAL;
	YPoint : LREAL;
END_VAR
END_METHOD

METHOD Build : I_PlanarTaskResult
END_METHOD

PROPERTY Busy : BOOL
GET
END_GET
END_PROPERTY

METHOD Clear : I_PlanarTaskResult
END_METHOD

METHOD CloseLoop : I_PlanarTaskResult
END_METHOD

{attribute 'hide'}
METHOD CyclicLogic
END_METHOD

{attribute 'suppress_wrn_C0410'}
PROPERTY Definition : REFERENCE TO ST_TrackDefinition
GET
END_GET
END_PROPERTY

METHOD Disable : I_PlanarTaskResult
END_METHOD

{attribute 'TcRpcEnable'}
METHOD Enable : I_PlanarTaskResult
END_METHOD

PROPERTY Error : BOOL
GET
END_GET
END_PROPERTY

PROPERTY ErrorId : UDINT
GET
END_GET
END_PROPERTY

METHOD GetTrackPositionAt : LREAL;
VAR_IN_OUT
	Position : PositionXYC;
END_VAR
END_METHOD

PROPERTY Index : UDINT
GET
END_GET
SET
END_SET
END_PROPERTY

{attribute 'hide'}
METHOD Initialize
END_METHOD

PROPERTY MoverCount : UDINT
GET
END_GET
END_PROPERTY

PROPERTY MovingMoverCount : UDINT
GET
END_GET
END_PROPERTY

{attribute 'suppress_wrn_C0410'}
PROPERTY pm : REFERENCE TO MC_PlanarTrack
GET
END_GET
END_PROPERTY

METHOD Reset : I_PlanarTaskResult
VAR_INPUT
END_VAR
END_METHOD

{attribute 'suppress_wrn_C0410'}
PROPERTY Status : REFERENCE TO CDT_MCTOPLC_PLANAR_TRACK
GET
END_GET
END_PROPERTY

PROPERTY TrackLength : LREAL
GET
END_GET
END_PROPERTY

PROPERTY Utility : I_McPlanarTrack
GET
END_GET
END_PROPERTY

END_INTERFACE

// _Internal/Movers/MoverQueue/FB_MoverQueue
FUNCTION_BLOCK FB_MoverQueue IMPLEMENTS I_MoverQueue
VAR
	MoversInQueue : UDINT := 0;
	ipMovers	  : ARRAY[1..Tc3_XPlanarUtility.Param_TcIoXPlanarEnvironment.MaxMcPlanarMovers] OF I_XPlanarMover;
END_VAR

//=============================================================================
//	Method Clear()
//=============================================================================
//
//	Brute force reset of buffer
//
//-----------------------------------------------------------------------------
METHOD Clear : BOOL
MEMSET(ADR(ipMovers), 0, SIZEOF(ipMovers));
MoversInQueue := 0;
Clear		  := TRUE;
END_METHOD

PROPERTY Count : UDINT
GET
VAR
	i	 : UDINT;
	temp : UDINT;
END_VAR
Count := MoversInQueue;
END_GET
END_PROPERTY

METHOD Dequeue : I_XPlanarMover
IF MoversInQueue > 0 THEN
	Dequeue := ipMovers[1];
	MEMSET(ADR(ipMovers[1]), 0, SIZEOF(ipMovers[1]));
	MoversInQueue := MoversInQueue - 1;
	IF MoversInQueue > 0 THEN
		MEMMOVE(ADR(ipMovers[1]), ADR(ipMovers[2]), SIZEOF(ipMovers[2]) * MoversInQueue);
		MEMSET(ADR(ipMovers[MoversInQueue + 1]), 0, (SIZEOF(ipMovers[1]) * (Tc3_XPlanarUtility.Param_TcIoXPlanarEnvironment.MaxMcPlanarMovers - MoversInQueue)));
	END_IF
END_IF
END_METHOD

METHOD Enqueue : BOOL
VAR_INPUT
	Mover : I_XPlanarMover;
END_VAR
VAR
	i : UDINT;
END_VAR
FOR i := 1 TO Tc3_XPlanarUtility.Param_TcIoXPlanarEnvironment.MaxMcPlanarMovers DO
	IF ipMovers[i] = Mover THEN		//Check if already in queue
		RETURN;
	ELSIF ipMovers[i] = 0 THEN		//Check if spot available
		ipMovers[i] := Mover;
		MoversInQueue := MoversInQueue + 1;
		Enqueue := TRUE;
		RETURN;
	END_IF
END_FOR
END_METHOD

PROPERTY FirstMover : I_XPlanarMover
GET
IF MoversInQueue > 0 THEN
	FirstMover := ipMovers[1];
END_IF
END_GET
END_PROPERTY

{attribute 'suppress_wrn_C0410'}
PROPERTY Queue : REFERENCE TO ARRAY[1..Tc3_XPlanarUtility.Param_TcIoXPlanarEnvironment.MaxMcPlanarMovers] OF I_XPlanarMover;
GET
VAR
	i : UDINT;
END_VAR
Queue ref= ipMovers;
END_GET
END_PROPERTY

END_FUNCTION_BLOCK

// _Internal/Movers/MoverQueue/I_MoverQueue
INTERFACE I_MoverQueue EXTENDS I_Base

//=============================================================================
//	Method Clear()
//=============================================================================
//
//	Brute force reset of buffer
//
//-----------------------------------------------------------------------------
METHOD Clear : BOOL
END_METHOD

PROPERTY Count : UDINT
GET
END_GET
END_PROPERTY

METHOD Dequeue : I_XPlanarMover
END_METHOD

METHOD Enqueue : BOOL
VAR_INPUT
	Mover : I_XPlanarMover;
END_VAR
END_METHOD

PROPERTY FirstMover : I_XPlanarMover
GET
END_GET
END_PROPERTY

{attribute 'suppress_wrn_C0410'}
PROPERTY Queue : REFERENCE TO ARRAY[1..Tc3_XPlanarUtility.Param_TcIoXPlanarEnvironment.MaxMcPlanarMovers] OF I_XPlanarMover;
GET
END_GET
END_PROPERTY

END_INTERFACE

// _Internal/NullObjects/FB_NullMover
{warning disable C0094}
FUNCTION_BLOCK FB_NullMover IMPLEMENTS I_XPlanarMover
VAR
END_VAR

PROPERTY ActualPosition : REFERENCE TO MoverVector
GET
END_GET
END_PROPERTY

METHOD AddToGroup : I_PlanarTaskResult
VAR_INPUT
	PlanarGroup	: REFERENCE TO MC_PlanarGroup;
END_VAR
END_METHOD

PROPERTY AtRotationPosition : BOOL
GET
END_GET
END_PROPERTY

PROPERTY Busy : BOOL
GET
END_GET
END_PROPERTY

PROPERTY CommandLog : REFERENCE TO ARRAY [0..SystemParameters.MAX_LOG_COUNT] OF ST_CommandLog
GET
END_GET
END_PROPERTY

METHOD CyclicLogic
END_METHOD

PROPERTY Destination : I_XPlanarStation
GET
END_GET
SET
END_SET
END_PROPERTY

METHOD Disable : I_PlanarTaskResult
END_METHOD

PROPERTY Dynamics : I_MoveDynamics
GET
END_GET
END_PROPERTY

METHOD Enable : I_PlanarTaskResult
END_METHOD

METHOD EnterMovementArea : I_PlanarTaskResult
VAR_INPUT
	PartId	: OTCID;
	PositionX	: LREAL;
	PositionY	: LREAL;
END_VAR
END_METHOD

PROPERTY Error : BOOL
GET
END_GET
END_PROPERTY

PROPERTY ErrorId : UDINT
GET
END_GET
END_PROPERTY

PROPERTY Gap : LREAL
GET
END_GET
SET
END_SET
END_PROPERTY

METHOD Halt : I_PlanarTaskResult
END_METHOD

PROPERTY IdentifiedBTN : STRING
GET
END_GET
SET
END_SET
END_PROPERTY

{attribute 'hide'}
METHOD Initialize
END_METHOD

PROPERTY InStation : BOOL
GET
END_GET
SET
END_SET
END_PROPERTY

PROPERTY LastCyclePosition : REFERENCE TO MoverVector
GET
END_GET
END_PROPERTY

METHOD LeaveMovementArea : I_PlanarTaskResult
END_METHOD

PROPERTY MoveCommand : I_MoveCommands
GET
END_GET
END_PROPERTY

PROPERTY MoverBTN : STRING
GET
END_GET
END_PROPERTY

PROPERTY MoverData : I_MoverData
GET
END_GET
SET
END_SET
END_PROPERTY

PROPERTY MoverIndex : UDINT
GET
END_GET
SET
END_SET
END_PROPERTY

PROPERTY MoverType : XplanarMoverType
GET
END_GET
SET
END_SET
END_PROPERTY

PROPERTY pm : REFERENCE TO MC_PlanarMover
GET
END_GET
END_PROPERTY

METHOD Reset : I_PlanarTaskResult
END_METHOD

PROPERTY RotationModulo : LREAL
GET
END_GET
END_PROPERTY

PROPERTY Status : REFERENCE TO CDT_MCTOPLC_PLANAR_MOVER_STD
GET
END_GET
END_PROPERTY

PROPERTY Utility : I_TcIoXPlanarMover
GET
END_GET
SET
END_SET
END_PROPERTY

END_FUNCTION_BLOCK

// _Internal/NullObjects/FB_NullMoverData
{warning disable C0094}
FUNCTION_BLOCK FB_NullMoverData IMPLEMENTS I_MoverData
VAR
END_VAR

END_FUNCTION_BLOCK

// _Internal/TaskBaseClasses/FB_MoverTask
{attribute 'no_explicit_call' := 'do not call this POU directly'}
FUNCTION_BLOCK FB_MoverTask EXTENDS FB_XPlanarTaskBase
VAR
	Mover		   : I_XPlanarMover;
	GetTime		   : GETSYSTEMTIME;
	SysTime		   : T_FILETIME;
	LogEntry	   : ST_MoverCommandInfo;
	ActualPosition : MoverVector;
	RT_ADSWarn	   : R_Trig;
	MoverStr	   : STRING;
END_VAR

METHOD CyclicLogic
ActualPosition := Mover.ActualPosition;
SUPER^.CyclicLogic();
RT_ADSWarn(CLK := _PlanarFb.Error);
IF RT_ADSWarn.Q THEN
	MoverStr := CONCAT('Mover ', TO_STRING(Mover.MoverIndex));
	LogEntry.Command := CONCAT(CONCAT(MoverStr, ' : %s'), CONCAT(LogEntry.Command, CONCAT('Error ', TO_STRING(_PlanarFb.ErrorId))));
	UpdateLog();
END_IF
END_METHOD

//FB_Init is always available implicitly and it is used primarily for initialization.
//The return value is not evaluated. For a specific influence, you can also declare the
//methods explicitly and provide additional code there with the standard initialization
//code. You can evaluate the return value.
METHOD FB_Init : BOOL
VAR_INPUT
	bInitRetains : BOOL; // TRUE: the retain variables are initialized (reset warm / reset cold)
	bInCopyCode	 : BOOL; // TRUE: the instance will be copied to the copy code afterward (online change)   
	Mover		 : I_XPlanarMover;
	Name		 : T_MaxString;
END_VAR
THIS^.Mover		:= Mover;
THIS^._TaskName := Name;
END_METHOD

METHOD UpdateLog
VAR_INST
	i : UINT;
END_VAR
IF SystemParameters.MAX_LOG_COUNT > 0 THEN
	FOR i := SystemParameters.MAX_LOG_COUNT - 1 TO 1 BY -1 DO
		IF i < SystemParameters.MAX_LOG_COUNT THEN
			Mover.CommandLog[i + 1] := Mover.CommandLog[i];
		END_IF
	END_FOR

	Mover.CommandLog[1] := Mover.CommandLog[0];
	GetTime(timeLoDW => SysTime.dwLowDateTime, timeHiDW => SysTime.dwHighDateTime);
	Mover.CommandLog[0].Timestamp := SYSTEMTIME_TO_STRING(FILETIME_TO_SYSTEMTIME(SysTime));
	Mover.CommandLog[0].Command	:= LogEntry.Command;
	Mover.CommandLog[0].Accel		:= LogEntry.Accel;
	Mover.CommandLog[0].Decel		:= LogEntry.Decel;
	Mover.CommandLog[0].Jerk		:= LogEntry.Jerk;
	Mover.CommandLog[0].Velocity	:= LogEntry.Velocity;
END_IF
END_METHOD

END_FUNCTION_BLOCK

// _Internal/TaskBaseClasses/FB_XPlanarTaskBase
{attribute 'no_assign_warning'}
{attribute 'no_explicit_call' := 'do not call this POU directly'}
FUNCTION_BLOCK FB_XPlanarTaskBase EXTENDS FB_TaskResult IMPLEMENTS I_Cyclic
VAR
	_PlanarFb		: MC_PlanarFeedback;
	HasRun			: BOOL;
	ExecuteWatchdog : UDINT;
	TaskState		: UDINT;
END_VAR

METHOD CyclicLogic
VAR_INST
	WatchdogCheck : UDINT;
END_VAR
//Update Command Feedback Status
_PlanarFb.Update();

//Update Interface based on Command Feedback status
_Aborted			:= _PlanarFb.Aborted;
_Busy				:= _PlanarFb.Active OR _PlanarFb.Busy;
_Done				:= _PlanarFb.Done;
_Error				:= _PlanarFb.Error;
_ErrorID			:= _PlanarFb.ErrorId;
_BlockingObjectInfo := _PlanarFb.objectInfo;

//Heartbeat to know execute is active
IF ExecuteWatchdog <> WatchdogCheck THEN
	WatchdogCheck := ExecuteWatchdog;
ELSE
	HasRun			:= FALSE;
	ExecuteWatchdog := 0;
END_IF
END_METHOD

{attribute 'suppress_wrn_C0410'}
PROPERTY PlanarFeedback : REFERENCE TO MC_PlanarFeedback
GET
PlanarFeedback ref= _PlanarFb;
END_GET
END_PROPERTY

END_FUNCTION_BLOCK

// _Internal/TaskBaseClasses/FB_TaskResult
{attribute 'no_explicit_call' := 'do not call this POU directly'}
FUNCTION_BLOCK FB_TaskResult IMPLEMENTS I_PlanarTaskResult
VAR
	_Busy				: BOOL;
	_Error				: BOOL;
	_ErrorID			: UDINT;
	_TaskName			: STRING;
	_Done				: BOOL;
	_Aborted			: BOOL;
	_BlockingObjectInfo : PlanarObjectInfo;
END_VAR

{attribute 'monitoring' := 'call'}
PROPERTY Aborted : BOOL
GET
Aborted := _Aborted;
END_GET
SET
_Aborted := Aborted;
END_SET
END_PROPERTY

{attribute 'suppress_wrn_C0410'}
PROPERTY BlockingObjectInfo : REFERENCE TO Tc3_Mc3PlanarMotion.PlanarObjectInfo
GET
BlockingObjectInfo ref= _BlockingObjectInfo;
END_GET
END_PROPERTY

{attribute 'monitoring' := 'call'}
PROPERTY Busy : BOOL
GET
Busy := _Busy;
END_GET
SET
_Busy := Busy;
END_SET
END_PROPERTY

{attribute 'monitoring' := 'call'}
PROPERTY Done : BOOL
GET
Done := _Done;
END_GET
SET
_Done := Done;
END_SET
END_PROPERTY

{attribute 'monitoring' := 'call'}
PROPERTY Error : BOOL
GET
Error := _Error;
END_GET
SET
_Error := Error;
END_SET
END_PROPERTY

{attribute 'monitoring' := 'call'}
PROPERTY ErrorID : UDINT
GET
ErrorID := _ErrorID;
END_GET
SET
_ErrorID := ErrorID;
END_SET
END_PROPERTY

PROPERTY Result : I_PlanarTaskResult
GET
Result := THIS^;
END_GET
END_PROPERTY

PROPERTY TaskName : STRING
GET
TaskName := _TaskName;
END_GET
SET
_TaskName := TaskName;
END_SET
END_PROPERTY

END_FUNCTION_BLOCK

// _Internal/TaskBaseClasses/FB_PartTask
{attribute 'no_explicit_call' := 'do not call this POU directly'}
FUNCTION_BLOCK FB_PartTask EXTENDS FB_XPlanarTaskBase
VAR
	ipPart : I_XplanarPart;
END_VAR

PROPERTY Part : I_XPlanarPart
SET
ipPart := Part;
END_SET
END_PROPERTY

END_FUNCTION_BLOCK

// Part/I_XPlanarPart
INTERFACE I_XPlanarPart EXTENDS __SYSTEM.IQueryInterface

PROPERTY Busy : BOOL
GET
END_GET
END_PROPERTY

PROPERTY Error : BOOL
GET
END_GET
END_PROPERTY

PROPERTY ErrorId : UDINT
GET
END_GET
END_PROPERTY

METHOD ForceDisable : I_PlanarTaskResult
END_METHOD

PROPERTY ObjectID : OTCID
GET
END_GET
END_PROPERTY

{attribute 'suppress_wrn_C0410'}
PROPERTY pm : REFERENCE TO MC_PlanarPart
GET
END_GET
END_PROPERTY

METHOD Reset : I_PlanarTaskResult
VAR_INPUT
END_VAR
END_METHOD

METHOD SetAllowEnable : I_PlanarTaskResult
END_METHOD

{attribute 'suppress_wrn_C0410'}
PROPERTY State : REFERENCE TO MC_PLANAR_STATE
GET
END_GET
END_PROPERTY

END_INTERFACE

// _Internal/TaskBaseClasses/FB_TrackTask
{attribute 'no_explicit_call' := 'do not call this POU directly'}
FUNCTION_BLOCK FB_TrackTask EXTENDS FB_XPlanarTaskBase
VAR
	ipTrack	   : I_XPlanarTrack;
END_VAR

PROPERTY Track : I_XplanarTrack
SET
ipTrack := Track;
END_SET
END_PROPERTY

END_FUNCTION_BLOCK

// Mover/TaskClasses/FB_AddToGroup
FUNCTION_BLOCK FB_AddToGroup EXTENDS FB_MoverTask
VAR
END_VAR

METHOD Execute : I_PlanarTaskResult
VAR_INPUT
	Group : REFERENCE TO MC_PlanarGroup;
END_VAR
IF NOT HasRun THEN
	_Done	 := FALSE;
	_Error	 := FALSE;
	_Busy	 := FALSE;
	_ErrorID := 0;
	Mover.pm.AddToGroup(_PlanarFb, Group);

	//Update mover command log				
	LogEntry.Command := CONCAT('AddMoverToGroup ', TO_STRING(Group.MCTOPLC_STD.GroupOID));
	LogEntry.Accel	 := 0;
	LogEntry.Decel	 := 0;
	LogEntry.Jerk	 := 0;
	LogEntry.Velocity := 0;
	UpdateLog();
	HasRun := TRUE;
END_IF

Execute := THIS^;

//Heartbeat that the method is active
ExecuteWatchdog := ExecuteWatchdog + 1;
END_METHOD

END_FUNCTION_BLOCK

// Mover/TaskClasses/FB_Disable
FUNCTION_BLOCK FB_Disable EXTENDS FB_MoverTask
VAR
END_VAR

METHOD Execute : I_PlanarTaskResult
VAR_INPUT
END_VAR
IF NOT HasRun AND Mover.Status.State <> MC_Planar_State.Disabled THEN
	_Done	 := FALSE;
	_Error	 := FALSE;
	_Busy	 := FALSE;
	_ErrorID := 0;
	Mover.pm.Disable(_PlanarFb);

	//Update mover command log				
	LogEntry.Command := 'DisableMover';
	LogEntry.Accel	 := 0;
	LogEntry.Decel	 := 0;
	LogEntry.Jerk	 := 0;
	LogEntry.Velocity := 0;
	UpdateLog();
	HasRun := TRUE;
END_IF

Execute := THIS^;

//Heartbeat that the method is active
ExecuteWatchdog := ExecuteWatchdog + 1;
END_METHOD

END_FUNCTION_BLOCK

// Mover/TaskClasses/FB_Enable
FUNCTION_BLOCK FB_Enable EXTENDS FB_MoverTask
VAR
END_VAR

METHOD Execute : I_PlanarTaskResult
IF NOT HasRun AND Mover.Status.State = MC_Planar_State.Disabled THEN
	_Done	 := FALSE;
	_Error	 := FALSE;
	_Busy	 := FALSE;
	_ErrorID := 0;
	Mover.pm.Enable(_PlanarFb);

	//Update mover command log				
	LogEntry.Command := 'EnableMover';
	LogEntry.Accel	 := 0;
	LogEntry.Decel	 := 0;
	LogEntry.Jerk	 := 0;
	LogEntry.Velocity := 0;
	UpdateLog();
	HasRun := TRUE;
END_IF

Execute := THIS^;

//Heartbeat that the method is active
ExecuteWatchdog := ExecuteWatchdog + 1;
END_METHOD

END_FUNCTION_BLOCK

// Mover/TaskClasses/FB_EnterMovementArea
FUNCTION_BLOCK FB_EnterMovementArea EXTENDS FB_MoverTask
VAR
	MovementAreaParameters : EnterOrLeaveMovementAreaParameters_XYC;
	EnterMvmtArea		   : BOOL;
END_VAR

METHOD CyclicLogic
VAR_INST
	WatchdogCheck : UDINT;
END_VAR
//State logic for the task
CASE TaskState OF
	0: // Init
		_Busy := FALSE;
		IF EnterMvmtArea THEN
			_Done		  := FALSE;
			_Error		  := FALSE;
			_ErrorID	  := 0;
			_Busy		  := TRUE;
			EnterMvmtArea := FALSE;
			TaskState	  := TaskState + 10;
		END_IF

	10: //Check input parameters
		IF MovementAreaParameters.MovementAreaOID = 0 OR MovementAreaParameters.Positions.x = 0 OR MovementAreaParameters.Positions.x = 0 THEN
			_Error	  := TRUE;
			_ErrorID  := 9999; //Invalid Entry
			TaskState := 0;
		ELSE
			TaskState := TaskState + 10;
		END_IF

	20: //Set Mover Movement Area
		IF Mover.Utility.SetMovementArea_XYC(MovementAreaParameters) THEN
			TaskState := TaskState + 10;
		END_IF

	30:
		IF SUCCEEDED(MovementAreaParameters.Result) THEN
			_Done	  := TRUE;
			TaskState := 0;
		ELSIF FAILED(MovementAreaParameters.Result) THEN
			_Error	  := TRUE;
			_ErrorID  := TO_UDINT(MovementAreaParameters.Result);
			TaskState := 0;
		END_IF
END_CASE

RT_ADSWarn(CLK := _Error);
IF RT_ADSWarn.Q THEN
	ADSLOGSTR(ADSLOG_MSGTYPE_WARN, CONCAT('Mover ', Mover.MoverBTN), CONCAT(_TaskName, CONCAT('Error ', TO_STRING(_ErrorId))));
END_IF

IF ExecuteWatchdog <> WatchdogCheck THEN
	WatchdogCheck := ExecuteWatchdog;
ELSE
	HasRun			:= FALSE;
	ExecuteWatchdog := 0;
END_IF
END_METHOD

METHOD Execute : I_PlanarTaskResult
VAR_INPUT
	PartId		: OTCID;
	PositionX	: LREAL;
	PositionY	: LREAL;
END_VAR
IF NOT HasRun THEN
	_Done								   := FALSE;
	_Error								   := FALSE;
	_Busy								   := FALSE;
	_ErrorID							   := 0;
	MovementAreaParameters.MovementAreaOID := PartId;
	MovementAreaParameters.Positions.x	   := PositionX;
	MovementAreaParameters.Positions.y	   := PositionY;
	EnterMvmtArea						   := TRUE;
	HasRun								   := TRUE;

	//Update mover command log				
	LogEntry.Command := CONCAT('Add To Movement Area', TO_STRING(PartId));
	UpdateLog();
END_IF

Execute := THIS^;

//Heartbeat that the method is active
ExecuteWatchdog := ExecuteWatchdog + 1;
END_METHOD

END_FUNCTION_BLOCK

// Mover/TaskClasses/FB_Halt
FUNCTION_BLOCK FB_Halt EXTENDS FB_MoverTask
VAR
	BusyStatus : MoverBusy;
END_VAR

METHOD Execute : I_PlanarTaskResult
VAR_INPUT
	Dynamics : REFERENCE TO DynamicConstraint_Coordinates;
END_VAR
BusyStatus := Mover.Status.Busy;
IF NOT HasRun AND BusyStatus.busyMover THEN
	_Done	 := FALSE;
	_Error	 := FALSE;
	_Busy	 := FALSE;
	_ErrorID := 0;
	Mover.pm.Halt(_PlanarFb, Dynamics);

	//Update mover command log				
	LogEntry.Command := 'HaltMover';
	UpdateLog();
	HasRun := TRUE;
END_IF

Execute := THIS^;

//Heartbeat that the method is active
ExecuteWatchdog := ExecuteWatchdog + 1;
END_METHOD

END_FUNCTION_BLOCK

// Mover/TaskClasses/FB_JoinClosestTrack
{attribute 'no_assign_warning'}
FUNCTION_BLOCK FB_JoinClosestTrack EXTENDS FB_MoverTask
VAR
	JoinTrackOptions	 : ST_JoinTrackOptions;
	TrackJoinDistances	 : ARRAY[1..Tc3_XPlanarUtility.Param_TcIoXPlanarEnvironment.MaxTracks] OF LREAL;
	_UseOrientation		 : BOOL;
	_MoveDynamics		 : DynamicConstraint_PathXYZ;
	i					 : UDINT;
	MoverSetPosition	 : MoverVector;
	MoverCurrentPosition : PositionXYC;
	MoverJoinPosition	 :  ARRAY[1..Tc3_XPlanarUtility.Param_TcIoXPlanarEnvironment.MaxTracks] OF PositionXYC;
	MoverArcPosition	 :  ARRAY[1..Tc3_XPlanarUtility.Param_TcIoXPlanarEnvironment.MaxTracks] OF LREAL;
	ShortestDistance	 : LREAL;
	TrackToJoin			 : UDINT;
	Join				 : BOOL;
END_VAR

METHOD CyclicLogic
VAR_INST
	WatchdogCheck : UDINT;
END_VAR
//***Overwriting the update method because this task contains a state machine that must be monitored cyclically.***
_PlanarFb.Update();

//State logic for the task
CASE TaskState OF
	0: // Init
		_Busy := FALSE;
		IF Join THEN
			_Done			 := FALSE;
			_Error			 := FALSE;
			_ErrorID		 := 0;
			_Busy			 := TRUE;
			Join			 := FALSE;
			ShortestDistance := 0;
			TaskState		 := TaskState + 10;
		END_IF

	10: //Resolve Mover Position
		MoverSetPosition	   := Mover.pm.MCTOPLC.SET.SetPos;
		MoverCurrentPosition.x := MoverSetPosition.x;
		MoverCurrentPosition.y := MoverSetPosition.y;
		MoverCurrentPosition.c := MoverSetPosition.c;
		TaskState			   := TaskState + 10;

	20: //Calculate distance from tracks
		FOR i := 1 TO XPlanar.TrackCount DO
			//Get arc position based on mover position
			MoverArcPosition[i] := ip.Tracks[i].GetTrackPositionAt(MoverCurrentPosition);

			//Get Position based on arc position
			ip.Tracks[i].pm.GetPositionAt(MoverArcPosition[i], MoverJoinPosition[i]);

			//Save position delta
			TrackJoinDistances[i] := ABS(MoverJoinPosition[i].x - MoverCurrentPosition.x) + ABS(MoverJoinPosition[i].y - MoverCurrentPosition.y);
		END_FOR

		TaskState := TaskState + 10;

	30: //Find Closest Track
		FOR i := 1 TO XPlanar.TrackCount DO
			IF ShortestDistance = 0 OR TrackJoinDistances[i] < ShortestDistance THEN
				ShortestDistance := TrackJoinDistances[i];
				TrackToJoin		 := i;
			END_IF
		END_FOR

		TaskState := TaskState + 10;

	40: //Join the closest track
		JoinTrackOptions.useOrientation := _UseOrientation;
		Mover.pm.JoinTrack(_PlanarFb,
							 ip.Tracks[TrackToJoin].pm,
							 _MoveDynamics,
							 JoinTrackOptions);

		//Update mover command log				
		LogEntry.Command := CONCAT('JoinClosestTrack : ', TO_STRING(TrackToJoin));
		LogEntry.Accel	 := _MoveDynamics.A;
		LogEntry.Decel	 := _MoveDynamics.D;
		LogEntry.Jerk	 := _MoveDynamics.J;
		LogEntry.Velocity := _MoveDynamics.V;
		UpdateLog();
		TaskState := TaskState + 10;

	50: //Watch feedback
		IF _PlanarFb.Done THEN
			TaskState := 60;
		ELSIF _PlanarFb.Error THEN
			_Error				:= TRUE;
			_ErrorID			:= _PlanarFb.ErrorId;
			_BlockingObjectInfo := _PlanarFb.objectInfo;
			TaskState			:= 0;
		END_IF

	60: //Task Complete
		THIS^._Done := TRUE;
		TaskState	:= 0;
END_CASE

RT_ADSWarn(CLK := _PlanarFb.Error);
IF RT_ADSWarn.Q THEN
	ADSLOGSTR(ADSLOG_MSGTYPE_WARN, CONCAT('Mover ', Mover.MoverBTN), CONCAT(_TaskName, CONCAT('Error ', TO_STRING(_PlanarFb.ErrorId))));
END_IF

IF ExecuteWatchdog <> WatchdogCheck THEN
	WatchdogCheck := ExecuteWatchdog;
ELSE
	HasRun			:= FALSE;
	ExecuteWatchdog := 0;
END_IF
END_METHOD

METHOD Execute : I_PlanarTaskResult
VAR_INPUT
	UseOrientation : BOOL;
	MoveDynamics   : DynamicConstraint_PathXYZ;
END_VAR
IF NOT HasRun AND (Mover.Status.CommandMode <> MC_Planar_Mover_Command_Mode.OnTrack) THEN
	_Done			:= FALSE;
	_Error			:= FALSE;
	_Busy			:= FALSE;
	_ErrorID		:= 0;
	_UseOrientation := UseOrientation;
	_MoveDynamics	:= MoveDynamics;
	Join			:= TRUE;
	HasRun			:= TRUE;
END_IF

Execute := THIS^;

//Heartbeat that the method is active
ExecuteWatchdog := ExecuteWatchdog + 1;
END_METHOD

END_FUNCTION_BLOCK

// Mover/TaskClasses/FB_JoinTrack
FUNCTION_BLOCK FB_JoinTrack EXTENDS FB_MoverTask
VAR
	JoinTrackOptions : ST_JoinTrackOptions;
END_VAR

METHOD Execute : I_PlanarTaskResult
VAR_INPUT
	ipTrack		   : I_XPlanarTrack;
	UseOrientation : BOOL;
	MoveDynamics   : REFERENCE TO DynamicConstraint_PathXYZ;
END_VAR
IF NOT HasRun AND (Mover.Status.CommandMode <> MC_Planar_Mover_Command_Mode.OnTrack) THEN
	_Done	 := FALSE;
	_Error	 := FALSE;
	_Busy	 := FALSE;
	_ErrorID := 0;
	JoinTrackOptions.useOrientation := UseOrientation;
	Mover.pm.JoinTrack(_PlanarFb,
					ipTrack.pm,
					MoveDynamics,
					JoinTrackOptions);

	//Update mover command log				
	LogEntry.Command := CONCAT('JoinTrack : ', TO_STRING(ipTrack.Index));
	LogEntry.Accel	 := MoveDynamics.A;
	LogEntry.Decel	 := MoveDynamics.D;
	LogEntry.Jerk	 := MoveDynamics.J;
	LogEntry.Velocity := MoveDynamics.V;
	UpdateLog();
	HasRun := TRUE;
END_IF

Execute := THIS^;

//Heartbeat that the method is active
ExecuteWatchdog := ExecuteWatchdog + 1;
END_METHOD

END_FUNCTION_BLOCK

// Mover/TaskClasses/FB_LeaveMovementArea
FUNCTION_BLOCK FB_LeaveMovementArea EXTENDS FB_MoverTask
VAR
	MovementAreaParameters : EnterOrLeaveMovementAreaParameters_XYC;
	LeaveMvmtArea		   : BOOL;
END_VAR

METHOD CyclicLogic
VAR_INST
	WatchdogCheck : UDINT;
END_VAR
//State logic for the task
CASE TaskState OF
	0: // Init
		_Busy := FALSE;
		IF LeaveMvmtArea THEN
			_Done		  := FALSE;
			_Error		  := FALSE;
			_ErrorID	  := 0;
			_Busy		  := TRUE;
			LeaveMvmtArea := FALSE;
			TaskState	  := TaskState + 10;
		END_IF

	10:  //Remove Mover from Movement Area
		IF Mover.Utility.SetMovementArea_XYC(MovementAreaParameters) THEN
			TaskState := TaskState + 10;
		END_IF

	20:
		IF SUCCEEDED(MovementAreaParameters.Result) THEN
			_Done	  := TRUE;
			TaskState := 0;
		ELSIF FAILED(MovementAreaParameters.Result) THEN
			_Error	  := TRUE;
			_ErrorID  := TO_UDINT(MovementAreaParameters.Result);
			TaskState := 0;
		END_IF
END_CASE

RT_ADSWarn(CLK := _Error);
IF RT_ADSWarn.Q THEN
	ADSLOGSTR(ADSLOG_MSGTYPE_WARN, CONCAT('Mover ', Mover.MoverBTN), CONCAT(_TaskName, CONCAT('Error ', TO_STRING(_ErrorId))));
END_IF

IF ExecuteWatchdog <> WatchdogCheck THEN
	WatchdogCheck := ExecuteWatchdog;
ELSE
	HasRun			:= FALSE;
	ExecuteWatchdog := 0;
END_IF
END_METHOD

METHOD Execute : I_PlanarTaskResult
IF NOT HasRun THEN
	_Done								   := FALSE;
	_Error								   := FALSE;
	_Busy								   := FALSE;
	_ErrorID							   := 0;
	MovementAreaParameters.MovementAreaOID := 0;
	LeaveMvmtArea						   := TRUE;
	HasRun								   := TRUE;

	//Update mover command log				
	LogEntry.Command := 'Remove From Movement Area';
	UpdateLog();
END_IF

Execute := THIS^;

//Heartbeat that the method is active
ExecuteWatchdog := ExecuteWatchdog + 1;
END_METHOD

END_FUNCTION_BLOCK

// Mover/TaskClasses/FB_LeaveTrack
{attribute 'no_assign_warning'}
FUNCTION_BLOCK FB_LeaveTrack EXTENDS FB_MoverTask
VAR
	LeaveTrackOptions : ST_LeaveTrackOptions;
END_VAR

METHOD Execute : I_PlanarTaskResult
VAR_INPUT
	TargetPositionX : LREAL;
	TargetPositionY : LREAL;
	UseOrientation	: BOOL;
	MoveDynamics	: REFERENCE TO DynamicConstraint_PathXYZ;
END_VAR

VAR_INST
	Target : PositionXYC;
END_VAR
IF NOT HasRun AND Mover.Status.CommandMode = MC_Planar_Mover_Command_Mode.OnTrack THEN
	_Done							 := FALSE;
	_Error							 := FALSE;
	_Busy							 := FALSE;
	_ErrorID						 := 0;
	LeaveTrackOptions.useOrientation := UseOrientation;
	Target.SetValuesXYC(TargetPositionX, TargetPositionY, ActualPosition.c);
	Mover.pm.LeaveTrack(_PlanarFb,
						  Target,
						  MoveDynamics,
						  LeaveTrackOptions);

	//Update mover command log				
	LogEntry.Command := CONCAT('LeaveTrackTo : ', CONCAT(CONCAT('X= ', TO_STRING(TargetPositionX)), CONCAT(' Y= ', TO_STRING(TargetPositionY))));
	LogEntry.Accel	 := MoveDynamics.A;
	LogEntry.Decel	 := MoveDynamics.D;
	LogEntry.Jerk	 := MoveDynamics.J;
	LogEntry.Velocity := MoveDynamics.V;
	UpdateLog();
	HasRun := TRUE;
END_IF

Execute := THIS^;

//Heartbeat that the method is active
ExecuteWatchdog := ExecuteWatchdog + 1;
END_METHOD

END_FUNCTION_BLOCK

// Mover/TaskClasses/FB_MoveA
FUNCTION_BLOCK FB_MoveA EXTENDS FB_MoverTask
VAR
	PositionBuffer	: LREAL;
END_VAR

METHOD Execute : I_PlanarTaskResult
VAR_INPUT
	Position	 : LREAL;
	MoveDynamics : REFERENCE TO DynamicConstraint_Coordinates;
END_VAR
IF NOT HasRun OR (Position <> PositionBuffer) THEN
	_Done	 := FALSE;
	_Error	 := FALSE;
	_Busy	 := FALSE;
	_ErrorID := 0;
	Mover.pm.MoveA(_PlanarFb, Position, MoveDynamics);

	//Update mover command log				
	LogEntry.Command := CONCAT('MoveA : ', TO_STRING(Position));
	LogEntry.Accel	 := MoveDynamics.GetA(Coord_Mcs_A1);
	LogEntry.Decel	 := MoveDynamics.GetD(Coord_Mcs_A1);
	LogEntry.Jerk	 := MoveDynamics.GetJ(Coord_Mcs_A1);
	LogEntry.Velocity := MoveDynamics.GetV(Coord_Mcs_A1);
	UpdateLog();
	
	//Update call buffers
	PositionBuffer := Position;
	HasRun := TRUE;
END_IF

Execute := THIS^;

//Heartbeat that the method is active
ExecuteWatchdog := ExecuteWatchdog + 1;
END_METHOD

END_FUNCTION_BLOCK

// Mover/TaskClasses/FB_MoveB
FUNCTION_BLOCK FB_MoveB EXTENDS FB_MoverTask
VAR
	PositionBuffer	: LREAL;
END_VAR

METHOD Execute : I_PlanarTaskResult
VAR_INPUT
	Position	 : LREAL;
	MoveDynamics : REFERENCE TO DynamicConstraint_Coordinates;
END_VAR
IF NOT HasRun OR (Position <> PositionBuffer) THEN
	_Done	 := FALSE;
	_Error	 := FALSE;
	_Busy	 := FALSE;
	_ErrorID := 0;
	Mover.pm.MoveB(_PlanarFb, Position, MoveDynamics);

	//Update mover command log				
	LogEntry.Command := CONCAT('MoveB : ', TO_STRING(Position));
	LogEntry.Accel	 := MoveDynamics.GetA(Coord_Mcs_B1);
	LogEntry.Decel	 := MoveDynamics.GetD(Coord_Mcs_B1);
	LogEntry.Jerk	 := MoveDynamics.GetJ(Coord_Mcs_B1);
	LogEntry.Velocity := MoveDynamics.GetV(Coord_Mcs_B1);
	UpdateLog();
	
	//Update call buffers
	PositionBuffer := Position;
	HasRun := TRUE;
END_IF

Execute := THIS^;

//Heartbeat that the method is active
ExecuteWatchdog := ExecuteWatchdog + 1;
END_METHOD

END_FUNCTION_BLOCK

// Mover/TaskClasses/FB_MoveRelativeC
FUNCTION_BLOCK FB_MoveRelativeC EXTENDS FB_MoverTask
VAR
	TargetBuffer	: LREAL;
END_VAR

METHOD Execute : I_PlanarTaskResult
VAR_INPUT
	Distance	 : LREAL;
	RotateDynamics : REFERENCE TO DynamicConstraint_Coordinates;
END_VAR
IF NOT HasRun OR (Distance <> TargetBuffer) THEN
	_Done	 := FALSE;
	_Error	 := FALSE;
	_Busy	 := FALSE;
	_ErrorID := 0;
	Mover.pm.MoveRelativeC(_PlanarFb, Distance, RotateDynamics);

	//Update mover command log				
	LogEntry.Command := CONCAT('MoveRelativeC : ', TO_STRING(Distance));
	LogEntry.Accel	 := RotateDynamics.GetA(Coord_Mcs_C1);
	LogEntry.Decel	 := RotateDynamics.GetD(Coord_Mcs_C1);
	LogEntry.Jerk	 := RotateDynamics.GetJ(Coord_Mcs_C1);
	LogEntry.Velocity := RotateDynamics.GetV(Coord_Mcs_C1);
	UpdateLog();
	
	//Update call buffers
	TargetBuffer := Distance;  //Keep track of last target position to let an updated command thru if in consecutive PLC cycles
	HasRun := TRUE; 
END_IF

Execute := THIS^;

//Heartbeat that the method is active
ExecuteWatchdog := ExecuteWatchdog + 1;
END_METHOD

END_FUNCTION_BLOCK

// Mover/TaskClasses/FB_MoveRelativeX
FUNCTION_BLOCK FB_MoveRelativeX EXTENDS FB_MoverTask
VAR
	TargetBuffer	: LREAL;
END_VAR

METHOD Execute : I_PlanarTaskResult
VAR_INPUT
	Distance	 : LREAL;
	MoveDynamics : REFERENCE TO DynamicConstraint_PathXYZ;
END_VAR
IF NOT HasRun OR (Distance <> TargetBuffer) THEN
	_Done	 := FALSE;
	_Error	 := FALSE;
	_Busy	 := FALSE;
	_ErrorID := 0;
	Mover.pm.MoveRelativeX(_PlanarFb, Distance, MoveDynamics);

	//Update mover command log				
	LogEntry.Command := CONCAT('MoveRelativeX : ', TO_STRING(Distance));
	LogEntry.Accel	 := MoveDynamics.A;
	LogEntry.Decel	 := MoveDynamics.D;
	LogEntry.Jerk	 := MoveDynamics.J;
	LogEntry.Velocity := MoveDynamics.V;
	UpdateLog();
	
	//Update call buffers
	TargetBuffer := Distance;  //Keep track of last target position to let an updated command thru if in consecutive PLC cycles
	HasRun := TRUE; 
END_IF

Execute := THIS^;

//Heartbeat that the method is active
ExecuteWatchdog := ExecuteWatchdog + 1;
END_METHOD

END_FUNCTION_BLOCK

// Mover/TaskClasses/FB_MoveRelativeY
FUNCTION_BLOCK FB_MoveRelativeY EXTENDS FB_MoverTask
VAR
	TargetBuffer	: LREAL;
END_VAR

METHOD Execute : I_PlanarTaskResult
VAR_INPUT
	Distance	 : LREAL;
	MoveDynamics : REFERENCE TO DynamicConstraint_PathXYZ;
END_VAR
IF NOT HasRun OR (Distance <> TargetBuffer) THEN
	_Done	 := FALSE;
	_Error	 := FALSE;
	_Busy	 := FALSE;
	_ErrorID := 0;
	Mover.pm.MoveRelativeY(_PlanarFb, Distance, MoveDynamics);

	//Update mover command log				
	LogEntry.Command := CONCAT('MoveRelativeY : ', TO_STRING(Distance));
	LogEntry.Accel	 := MoveDynamics.A;
	LogEntry.Decel	 := MoveDynamics.D;
	LogEntry.Jerk	 := MoveDynamics.J;
	LogEntry.Velocity := MoveDynamics.V;
	UpdateLog();
	
	//Update call buffers
	TargetBuffer := Distance;  //Keep track of last target position to let an updated command thru if in consecutive PLC cycles
	HasRun := TRUE; 
END_IF

Execute := THIS^;

//Heartbeat that the method is active
ExecuteWatchdog := ExecuteWatchdog + 1;
END_METHOD

END_FUNCTION_BLOCK

// Mover/TaskClasses/FB_MoveToPosition
{attribute 'no_assign_warning'}
FUNCTION_BLOCK FB_MoveToPosition EXTENDS FB_MoverTask
VAR
	MoveOptions		: ST_MoveToPositionOptions;
	MoverPosition	: MoverVector;
	Position		: PositionXYC;
	XPositionBuffer : LREAL;
	YPositionBuffer : LREAL;
END_VAR

METHOD Execute : I_PlanarTaskResult
VAR_INPUT
	XTarget		  : LREAL;
	YTarget		  : LREAL;
	CTarget		  : LREAL;

	MoveDynamics  : REFERENCE TO DynamicConstraint_PathXYZ;
		Rototranslate : BOOL := FALSE;
END_VAR
IF NOT HasRun OR ((XTarget <> XPositionBuffer) OR (YTarget <> YPositionBuffer)) THEN
	_Done	 := FALSE;
	_Error	 := FALSE;
	_Busy	 := FALSE;
	_ErrorID := 0;
	
	//Check for rototranslation
	IF Rototranslate THEN
		MoverPosition.c := CTarget;
	ELSE
		MoverPosition := Mover.pm.MCTOPLC.SET.SetPos;
	END_IF

	//Move Command
	Position.SetValuesXYC(XTarget, YTarget, MoverPosition.c);
	Mover.pm.MoveToPosition(_PlanarFb,
							Position,
							MoveDynamics,
							MoveOptions);

	//Update mover command log				
	LogEntry.Command  := CONCAT('MoveToPosition : ', CONCAT(CONCAT('X= ', TO_STRING(XTarget)), CONCAT(' Y= ', TO_STRING(YTarget))));
	LogEntry.Accel	  := MoveDynamics.A;
	LogEntry.Decel	  := MoveDynamics.D;
	LogEntry.Jerk	  := MoveDynamics.J;
	LogEntry.Velocity := MoveDynamics.V;
	UpdateLog();

	//Update call buffers
	XPositionBuffer := XTarget;
	YPositionBuffer := YTarget;
	HasRun			:= TRUE;
END_IF

//Return interface for status
Execute := THIS^;

//Heartbeat that the method is active
ExecuteWatchdog := ExecuteWatchdog + 1;
END_METHOD

END_FUNCTION_BLOCK

// Mover/TaskClasses/FB_MoveVelocityC
FUNCTION_BLOCK FB_MoveVelocityC EXTENDS FB_MoverTask
VAR
	TargetBuffer	: LREAL;
END_VAR

METHOD Execute : I_PlanarTaskResult
VAR_INPUT
	Velocity	 : LREAL;
	RotateDynamics : REFERENCE TO DynamicConstraint_Coordinates;
END_VAR
IF NOT HasRun OR (Velocity <> TargetBuffer) THEN
	_Done	 := FALSE;
	_Error	 := FALSE;
	_Busy	 := FALSE;
	_ErrorID := 0;
	Mover.pm.MoveVelocityC(_PlanarFb, Velocity, RotateDynamics);

	//Update mover command log				
	LogEntry.Command := CONCAT('MoveVelocityC : ', TO_STRING(Velocity));
	LogEntry.Accel	 := RotateDynamics.GetA(Coord_Mcs_C1);
	LogEntry.Decel	 := RotateDynamics.GetD(Coord_Mcs_C1);
	LogEntry.Jerk	 := RotateDynamics.GetJ(Coord_Mcs_C1);
	LogEntry.Velocity := RotateDynamics.GetV(Coord_Mcs_C1);
	UpdateLog();
	
	//Update call buffers
	TargetBuffer := Velocity;  //Keep track of last target position to let an updated command thru if in consecutive PLC cycles
	HasRun := TRUE; 
END_IF

Execute := THIS^;

//Heartbeat that the method is active
ExecuteWatchdog := ExecuteWatchdog + 1;
END_METHOD

END_FUNCTION_BLOCK

// Mover/TaskClasses/FB_MoveVelocityX
FUNCTION_BLOCK FB_MoveVelocityX EXTENDS FB_MoverTask
VAR
	TargetBuffer	: LREAL;
END_VAR

METHOD Execute : I_PlanarTaskResult
VAR_INPUT
	Velocity	 : LREAL;
	MoveDynamics : REFERENCE TO DynamicConstraint_PathXYZ;
END_VAR
IF NOT HasRun OR (Velocity <> TargetBuffer) THEN
	_Done	 := FALSE;
	_Error	 := FALSE;
	_Busy	 := FALSE;
	_ErrorID := 0;
	Mover.pm.MoveVelocityX(_PlanarFb, Velocity, MoveDynamics);

	//Update mover command log				
	LogEntry.Command := CONCAT('MoveVelocityX : ', TO_STRING(Velocity));
	LogEntry.Accel	 := MoveDynamics.A;
	LogEntry.Decel	 := MoveDynamics.D;
	LogEntry.Jerk	 := MoveDynamics.J;
	LogEntry.Velocity := MoveDynamics.V;
	UpdateLog();
	
	//Update call buffers
	TargetBuffer := Velocity;  //Keep track of last target position to let an updated command thru if in consecutive PLC cycles
	HasRun := TRUE; 
END_IF

Execute := THIS^;

//Heartbeat that the method is active
ExecuteWatchdog := ExecuteWatchdog + 1;
END_METHOD

END_FUNCTION_BLOCK

// Mover/TaskClasses/FB_MoveVelocityY
FUNCTION_BLOCK FB_MoveVelocityY EXTENDS FB_MoverTask
VAR
	TargetBuffer	: LREAL;
END_VAR

METHOD Execute : I_PlanarTaskResult
VAR_INPUT
	Velocity	 : LREAL;
	MoveDynamics : REFERENCE TO DynamicConstraint_PathXYZ;
END_VAR
IF NOT HasRun OR (Velocity <> TargetBuffer) THEN
	_Done	 := FALSE;
	_Error	 := FALSE;
	_Busy	 := FALSE;
	_ErrorID := 0;
	Mover.pm.MoveVelocityY(_PlanarFb, Velocity, MoveDynamics);

	//Update mover command log				
	LogEntry.Command := CONCAT('MoveVelocityY : ', TO_STRING(Velocity));
	LogEntry.Accel	 := MoveDynamics.A;
	LogEntry.Decel	 := MoveDynamics.D;
	LogEntry.Jerk	 := MoveDynamics.J;
	LogEntry.Velocity := MoveDynamics.V;
	UpdateLog();
	
	//Update call buffers
	TargetBuffer := Velocity;  //Keep track of last target position to let an updated command thru if in consecutive PLC cycles
	HasRun := TRUE; 
END_IF

Execute := THIS^;

//Heartbeat that the method is active
ExecuteWatchdog := ExecuteWatchdog + 1;
END_METHOD

END_FUNCTION_BLOCK

// Mover/TaskClasses/FB_MoveX
FUNCTION_BLOCK FB_MoveX EXTENDS FB_MoverTask
VAR
	PositionBuffer	: LREAL;
END_VAR

METHOD Execute : I_PlanarTaskResult
VAR_INPUT
	Position	 : LREAL;
	MoveDynamics : REFERENCE TO DynamicConstraint_PathXYZ;
END_VAR
IF NOT HasRun OR (Position <> PositionBuffer) THEN
	_Done	 := FALSE;
	_Error	 := FALSE;
	_Busy	 := FALSE;
	_ErrorID := 0;
	Mover.pm.MoveX(_PlanarFb, Position, 0, MoveDynamics);
	
	//Update mover command log				
	LogEntry.Command := CONCAT('MoveX : ', TO_STRING(Position));
	LogEntry.Accel	 := MoveDynamics.A;
	LogEntry.Decel	 := MoveDynamics.D;
	LogEntry.Jerk	 := MoveDynamics.J;
	LogEntry.Velocity := MoveDynamics.V;
	UpdateLog();
	
	//Update call buffers
	PositionBuffer := Position;  //Keep track of last target position to let an updated command thru if in consecutive PLC cycles
	HasRun := TRUE; 
END_IF

Execute := THIS^;

//Heartbeat that the method is active
ExecuteWatchdog := ExecuteWatchdog + 1;
END_METHOD

END_FUNCTION_BLOCK

// Mover/TaskClasses/FB_MoveY
FUNCTION_BLOCK FB_MoveY EXTENDS FB_MoverTask
VAR
	PositionBuffer	: LREAL;
END_VAR

METHOD Execute : I_PlanarTaskResult
VAR_INPUT
	Position	 : LREAL;
	MoveDynamics : REFERENCE TO DynamicConstraint_PathXYZ;
END_VAR
IF NOT HasRun OR (Position <> PositionBuffer) THEN
	_Done	 := FALSE;
	_Error	 := FALSE;
	_Busy	 := FALSE;
	_ErrorID := 0;
	Mover.pm.MoveY(_PlanarFb, Position, 0, MoveDynamics);

	//Update mover command log				
	LogEntry.Command := CONCAT('MoveY : ', TO_STRING(Position));
	LogEntry.Accel	 := MoveDynamics.A;
	LogEntry.Decel	 := MoveDynamics.D;
	LogEntry.Jerk	 := MoveDynamics.J;
	LogEntry.Velocity := MoveDynamics.V;
	UpdateLog();
	
	//Update call buffers
	PositionBuffer := Position;  //Keep track of last target position to let an updated command thru if in consecutive PLC cycles
	HasRun := TRUE; 
END_IF

Execute := THIS^;

//Heartbeat that the method is active
ExecuteWatchdog := ExecuteWatchdog + 1;
END_METHOD

END_FUNCTION_BLOCK

// Mover/TaskClasses/FB_MoveZ
FUNCTION_BLOCK FB_MoveZ EXTENDS FB_MoverTask
VAR
	PositionBuffer	: LREAL;
END_VAR

METHOD Execute : I_PlanarTaskResult
VAR_INPUT
	Position	 : LREAL;
	MoveDynamics : REFERENCE TO DynamicConstraint_PathXYZ;
END_VAR
IF NOT HasRun OR (Position <> PositionBuffer) THEN
	_Done	 := FALSE;
	_Error	 := FALSE;
	_Busy	 := FALSE;
	_ErrorID := 0;
	Mover.pm.MoveZ(_PlanarFb, Position, MoveDynamics);

	//Update mover command log				
	LogEntry.Command := CONCAT('MoveZ : ', TO_STRING(Position));
	LogEntry.Accel	 := MoveDynamics.A;
	LogEntry.Decel	 := MoveDynamics.D;
	LogEntry.Jerk	 := MoveDynamics.J;
	LogEntry.Velocity := MoveDynamics.V;
	UpdateLog();
	
	//Update call buffers
	PositionBuffer := Position;  //Keep track of last target position to let an updated command thru if in consecutive PLC cycles
	HasRun := TRUE; 
END_IF

Execute := THIS^;

//Heartbeat that the method is active
ExecuteWatchdog := ExecuteWatchdog + 1;
END_METHOD

END_FUNCTION_BLOCK

// Mover/TaskClasses/FB_ResetMover
FUNCTION_BLOCK FB_ResetMover EXTENDS FB_MoverTask
VAR
END_VAR

METHOD Execute : I_PlanarTaskResult
IF NOT HasRun THEN
	_Done		:= FALSE;
	_Error		:= FALSE;
	_Busy		:= FALSE;
	_ErrorID	:= 0;
	Mover.pm.Reset(_PlanarFb);
	HasRun := TRUE;
END_IF

Execute := THIS^;

//Heartbeat that the method is active
ExecuteWatchdog := ExecuteWatchdog + 1;
END_METHOD

END_FUNCTION_BLOCK

// Mover/TaskClasses/FB_Rotate
FUNCTION_BLOCK FB_Rotate EXTENDS FB_MoverTask
VAR
	RotateOptions : ST_MoveCOptions;
	PositionBuffer	: LREAL;
	TurnsBuffer		: DINT;
END_VAR

METHOD Execute : I_PlanarTaskResult
VAR_INPUT
	Distance	   : LREAL;
	NumberOfTurns  : DINT;
	Direction	   : Tc3_Mc3PlanarMotion.MC_DIRECTION;
	RotateDynamics : REFERENCE TO DynamicConstraint_Coordinates;
END_VAR
IF NOT HasRun OR ((Distance <> PositionBuffer) OR (NumberOfTurns <> TurnsBuffer)) THEN
	_Done						  := FALSE;
	_Error						  := FALSE;
	_Busy						  := FALSE;
	_ErrorID					  := 0;
	RotateOptions.direction		  := Direction;
	RotateOptions.additionalTurns := TO_UDINT(NumberOfTurns);
	Mover.pm.MoveC(_PlanarFb,
					 Distance,
					 RotateDynamics,
					 RotateOptions);

	//Update mover command log				
	LogEntry.Command := CONCAT('MoveC : ', CONCAT(TO_STRING(Distance), CONCAT(' : Turns ', TO_STRING(NumberOfTurns))));
	LogEntry.Accel	 := RotateDynamics.GetA(Coord_Mcs_C1);
	LogEntry.Decel	 := RotateDynamics.GetD(Coord_Mcs_C1);
	LogEntry.Jerk	 := RotateDynamics.GetJ(Coord_Mcs_C1);
	LogEntry.Velocity := RotateDynamics.GetV(Coord_Mcs_C1);
	UpdateLog();

	//Update call buffers
	PositionBuffer := Distance;
	TurnsBuffer	   := NumberOfTurns;
	HasRun		   := TRUE;
END_IF

Execute := THIS^;

//Heartbeat that the method is active
ExecuteWatchdog := ExecuteWatchdog + 1;
END_METHOD

END_FUNCTION_BLOCK

// Mover/TaskClasses/FB_RunExternalSetpointAbsoluteMode
FUNCTION_BLOCK FB_RunExternalSetpointAbsoluteMode EXTENDS FB_MoverTask
VAR
	ExternalSetpointGenerationOptions : ST_ExternalSetpointGenerationOptions;
END_VAR

METHOD Execute : I_PlanarTaskResult
VAR_INPUT
	Position	 : MoverVector;
	Velocity	 : MoverVector;
	Acceleration : MoverVector;
END_VAR
IF NOT HasRun THEN
	_Done								   := FALSE;
	_Error								   := FALSE;
	_Busy								   := FALSE;
	_ErrorID							   := 0;
	ExternalSetpointGenerationOptions.mode := MC_EXTERNAL_SET_POSITION_MODE.Absolute;
	Mover.pm.StartExternalSetpointGeneration(_PlanarFb, ExternalSetpointGenerationOptions);

	//Update mover command log				
	LogEntry.Command := CONCAT('Follow External setpoint started at : ', CONCAT(CONCAT('X= ', TO_STRING(Position.x)), CONCAT(' Y= ', TO_STRING(Position.y))));
	UpdateLog();
	HasRun := TRUE;
END_IF

Mover.pm.SetExternalSetpoint(Position, Velocity, Acceleration);
Execute := THIS^;

//Heartbeat that the method is active
ExecuteWatchdog := ExecuteWatchdog + 1;
END_METHOD

END_FUNCTION_BLOCK

// Mover/TaskClasses/FB_RunExternalSetpointRelativeMode
FUNCTION_BLOCK FB_RunExternalSetpointRelativeMode EXTENDS FB_MoverTask
VAR
	ExternalSetpointGenerationOptions : ST_ExternalSetpointGenerationOptions;
END_VAR

METHOD Execute : I_PlanarTaskResult
VAR_INPUT
	Position	 : MoverVector;
	Velocity	 : MoverVector;
	Acceleration : MoverVector;
END_VAR
IF NOT HasRun THEN
	_Done								   := FALSE;
	_Error								   := FALSE;
	_Busy								   := FALSE;
	_ErrorID							   := 0;
	ExternalSetpointGenerationOptions.mode := MC_EXTERNAL_SET_POSITION_MODE.Relative;
	Mover.pm.StartExternalSetpointGeneration(_PlanarFb, ExternalSetpointGenerationOptions);

	//Update mover command log				
	LogEntry.Command := CONCAT('Follow External setpoint started at : ', CONCAT(CONCAT('X= ', TO_STRING(Position.x)), CONCAT(' Y= ', TO_STRING(Position.y))));
	UpdateLog();
	HasRun := TRUE;
END_IF

Mover.pm.SetExternalSetpoint(Position, Velocity, Acceleration);
Execute := THIS^;

//Heartbeat that the method is active
ExecuteWatchdog := ExecuteWatchdog + 1;
END_METHOD

END_FUNCTION_BLOCK

// Mover/TaskClasses/FB_SquareUp
{attribute 'no_assign_warning'} 
FUNCTION_BLOCK FB_SquareUp EXTENDS FB_MoverTask
VAR
	RotateOptions	: Tc3_Mc3PlanarMotion.ST_MoveCOptions;
	_RotateDynamics : REFERENCE TO Tc3_Physics.DynamicConstraint_Coordinates;
	_MoveDynamics	: REFERENCE TO Tc3_Physics.DynamicConstraint_PathXYZ;
	_Distance		: LREAL;
	SquareUp		: BOOL;
END_VAR

METHOD CyclicLogic
VAR_INST
	WatchdogCheck : UDINT;
END_VAR
//***Overwriting the update method because this task contains a state machine that must be monitored cyclically.***
_PlanarFb.Update();

//State logic for the task
CASE TaskState OF
	0: // Init
		_Busy := FALSE;
		IF SquareUp THEN
			_Done	  := FALSE;
			_Error	  := FALSE;
			_Aborted  := FALSE;
			_ErrorID  := 0;
			_Busy	  := TRUE;
			SquareUp  := FALSE;
			TaskState := TaskState + 10;
		END_IF

	10: //Rotate C to closest quarter angle
		RotateOptions.direction		  := Tc3_Mc3PlanarMotion.MC_DIRECTION.mcDirectionShortestWay;
		RotateOptions.additionalTurns := 0;
		Mover.pm.MoveC(_PlanarFb,
						 _Distance,
						 _RotateDynamics,
						 RotateOptions);

		//Update mover command log				
		LogEntry.Command := CONCAT('MoveC : ', TO_STRING(_Distance));
		LogEntry.Accel	 := _RotateDynamics.GetA(Coord_Mcs_C1);
		LogEntry.Decel	 := _RotateDynamics.GetD(Coord_Mcs_C1);
		LogEntry.Jerk	 := _RotateDynamics.GetJ(Coord_Mcs_C1);
		LogEntry.Velocity := _RotateDynamics.GetV(Coord_Mcs_C1);
		UpdateLog();
		TaskState := TaskState + 10;

	20: //Watch rotate feedback
		IF _PlanarFb.Done THEN
			TaskState := TaskState + 10;
		ELSIF _PlanarFb.Error THEN
			TaskState := 999;
		ELSIF _PlanarFb.Aborted THEN
			_Aborted  := TRUE;
			TaskState := 0;
		END_IF

	30: //Move A Axis to 0
		Mover.pm.MoveA(_PlanarFb, 0.0, _MoveDynamics);

		//Update mover command log				
		LogEntry.Command := CONCAT('Move A : ', TO_STRING(0.0));
		LogEntry.Accel	 := _MoveDynamics.A;
		LogEntry.Decel	 := _MoveDynamics.D;
		LogEntry.Jerk	 := _MoveDynamics.J;
		LogEntry.Velocity := _MoveDynamics.V;
		UpdateLog();
		TaskState := TaskState + 10;

	40: //A Axis move feedback
		IF _PlanarFb.Done THEN
			TaskState := TaskState + 10;
		ELSIF _PlanarFb.Error THEN
			TaskState := 999;
		ELSIF _PlanarFb.Aborted THEN
			_Aborted := TRUE;
			TaskState := 0;
		END_IF

	50: //Move B Axis to 0
		Mover.pm.MoveB(_PlanarFb, 0.0, _MoveDynamics);

		//Update mover command log				
		LogEntry.Command := CONCAT('Move B : ', TO_STRING(0.0));
		LogEntry.Accel	 := _MoveDynamics.A;
		LogEntry.Decel	 := _MoveDynamics.D;
		LogEntry.Jerk	 := _MoveDynamics.J;
		LogEntry.Velocity := _MoveDynamics.V;
		UpdateLog();
		TaskState := TaskState + 10;

	60: //A Axis move feedback
		IF _PlanarFb.Done THEN
			TaskState := TaskState + 10;
		ELSIF _PlanarFb.Error THEN
			TaskState := 999;
		ELSIF _PlanarFb.Aborted THEN
			_Aborted := TRUE;
			TaskState := 0;
		END_IF

	70: //Task Complete
		_Done	  := TRUE;
		TaskState := 0;

	999: //Task Error
		_Error				:= TRUE;
		_ErrorID			:= _PlanarFb.ErrorId;
		_BlockingObjectInfo := _PlanarFb.objectInfo;
		TaskState			:= 0;
END_CASE

IF TaskState > 0 AND Mover.Error THEN
	TaskState := 999;
END_IF

IF ExecuteWatchdog <> WatchdogCheck THEN
	WatchdogCheck := ExecuteWatchdog;
ELSE
	HasRun			:= FALSE;
	ExecuteWatchdog := 0;
END_IF
END_METHOD

METHOD Execute : I_PlanarTaskResult
VAR_INPUT
	Distance	   : LREAL;
	RotateDynamics : REFERENCE TO Tc3_Physics.DynamicConstraint_Coordinates;
	MoveDynamics   : REFERENCE TO Tc3_Physics.DynamicConstraint_PathXYZ;
END_VAR
IF NOT HasRun THEN
	_Done			:= FALSE;
	_Error			:= FALSE;
	_Busy			:= FALSE;
	_ErrorID		:= 0;
	_Distance		:= Distance;
	_RotateDynamics REF= RotateDynamics;
	_MoveDynamics	ref= MoveDynamics;
	SquareUp		:= TRUE;
	HasRun			:= TRUE;
END_IF

Execute := THIS^;

//Heartbeat that the method is active
ExecuteWatchdog := ExecuteWatchdog + 1;
END_METHOD

END_FUNCTION_BLOCK

// Mover/TaskClasses/FB_StopExternalSetpoint
FUNCTION_BLOCK FB_StopExternalSetpoint EXTENDS FB_MoverTask
VAR
	ExternalSetpointGenerationOptions : ST_ExternalSetpointGenerationOptions;
END_VAR

METHOD Execute : I_PlanarTaskResult
IF NOT HasRun THEN
	_Done	 := FALSE;
	_Error	 := FALSE;
	_Busy	 := FALSE;
	_ErrorID := 0;
	Mover.pm.StopExternalSetpointGeneration(_PlanarFb);

	//Update mover command log				
	LogEntry.Command := 'Stop external setpoint';
	UpdateLog();
	HasRun := TRUE;
END_IF

Execute := THIS^;

//Heartbeat that the method is active
ExecuteWatchdog := ExecuteWatchdog + 1;
END_METHOD

END_FUNCTION_BLOCK

// Mover/TaskClasses/FB_TrackMove
{attribute 'no_assign_warning'} 
FUNCTION_BLOCK FB_TrackMove EXTENDS FB_MoverTask
VAR
	DynMove			   : DynamicConstraint_PathXY;
	MoveOnTrackOptions : ST_MoveOnTrackOptions;
	MoverSetPos		   : MoverVector;
	OnTrackPos		   : LREAL;
END_VAR

METHOD Execute : I_PlanarTaskResult
VAR_INPUT
	Position	 : LREAL;
	Gap			 : LREAL;
	TrackSegment : I_XPlanarTrack;
	MoveDynamics : REFERENCE TO DynamicConstraint_PathXY;
	Direction	 : Tc3_Mc3PlanarMotion.MC_DIRECTION;
END_VAR
IF NOT HasRun AND (Mover.Status.CommandMode = MC_Planar_Mover_Command_Mode.OnTrack OR Mover.Status.CommandMode = MC_Planar_Mover_Command_Mode.CRotationOnTrack) THEN
	_Done		:= FALSE;
	_Error		:= FALSE;
	_Busy		:= FALSE;
	_ErrorID	:= 0;
	MoveOnTrackOptions.gap		 := Gap;
	MoveOnTrackOptions.direction := Direction;
	
	IF SystemParameters.AutoDynamicsReduction THEN
		MoveOnTrackOptions.dynamicMode := MC_DYNAMICS_REDUCTION_MODE.AccelerationLimitedVelocity;
	ELSE
		MoveOnTrackOptions.dynamicMode := MC_DYNAMICS_REDUCTION_MODE.None;
	END_IF
	
	Mover.pm.MoveOnTrack(_PlanarFb,
					  TrackSegment.pm,
					  Position,
					  MoveDynamics,
					  MoveOnTrackOptions);

	//Update mover command log				
	LogEntry.Command := CONCAT('MoveOnTrack : ', CONCAT(CONCAT('ID : ', TO_STRING(TrackSegment.Index)), CONCAT(' Pos ', TO_STRING(Position))));
	LogEntry.Accel	 := MoveDynamics.A;
	LogEntry.Decel	 := MoveDynamics.D;
	LogEntry.Jerk	 := MoveDynamics.J;
	LogEntry.Velocity := MoveDynamics.V;
	UpdateLog();
	HasRun := TRUE;
END_IF

Execute := THIS^;

//Heartbeat that the method is active
ExecuteWatchdog := ExecuteWatchdog + 1;
END_METHOD

END_FUNCTION_BLOCK

// Mover/TaskClasses/FB_TrackMoveXY
{attribute 'no_assign_warning'}
FUNCTION_BLOCK FB_TrackMoveXY EXTENDS FB_MoverTask
VAR
	DynMove			   : DynamicConstraint_PathXY;
	MoveOnTrackOptions : ST_MoveOnTrackOptions;
END_VAR

METHOD Execute : I_PlanarTaskResult
VAR_INPUT
	PositionX	 : LREAL;
	PositionY	 : LREAL;
	Gap			 : LREAL;
	TrackSegment : I_XPlanarTrack;
	MoveDynamics : REFERENCE TO DynamicConstraint_PathXY;
	Direction	 : Tc3_Mc3PlanarMotion.MC_DIRECTION;
END_VAR

VAR_INST
	Position		: PositionXYC;
	SetPosition		: MoverVector;
	OnTrackPosition : LREAL;
END_VAR
IF NOT HasRun AND (Mover.Status.CommandMode = MC_Planar_Mover_Command_Mode.OnTrack OR Mover.Status.CommandMode = MC_Planar_Mover_Command_Mode.CRotationOnTrack) THEN
	_Done		:= FALSE;
	_Error		:= FALSE;
	_Busy		:= FALSE;
	_ErrorID	:= 0;
	SetPosition := Mover.pm.MCTOPLC.SET.SetPos;
	Position.SetValuesXY(PositionX, PositionY);
	MoveOnTrackOptions.gap		 := Gap;
	MoveOnTrackOptions.direction := Direction;
	
	IF SystemParameters.AutoDynamicsReduction THEN
		MoveOnTrackOptions.dynamicMode := MC_DYNAMICS_REDUCTION_MODE.AccelerationLimitedVelocity;
	ELSE
		MoveOnTrackOptions.dynamicMode := MC_DYNAMICS_REDUCTION_MODE.None;
	END_IF

	OnTrackPosition := TrackSegment.GetTrackPositionAt(Position);
	Mover.pm.MoveOnTrack(_PlanarFb,
						 TrackSegment.pm,
						 OnTrackPosition,
						 MoveDynamics,
						 MoveOnTrackOptions);

	//Update mover command log				
		LogEntry.Command := CONCAT('MoveOnTrack : ', CONCAT(CONCAT('ID : ', TO_STRING(TrackSegment.Index)), CONCAT(' Pos ', TO_STRING(OnTrackPosition))));

	LogEntry.Accel	  := MoveDynamics.A;
	LogEntry.Decel	  := MoveDynamics.D;
	LogEntry.Jerk	  := MoveDynamics.J;
	LogEntry.Velocity := MoveDynamics.V;
	UpdateLog();
	HasRun := TRUE;
END_IF

Execute := THIS^;

//Heartbeat that the method is active
ExecuteWatchdog := ExecuteWatchdog + 1;
END_METHOD

END_FUNCTION_BLOCK

// Mover/FB_XPlanarMover
{attribute 'no_assign'}
{attribute 'no_explicit_call' := 'do not call this POU directly'}
FUNCTION_BLOCK FB_XPlanarMover IMPLEMENTS I_Cyclic, I_Initializable, I_XPlanarMover, I_MoveCommands, I_MoveDynamics
VAR
	//Planar Motion Vars
	_Mover		: Tc3_MC3PlanarMotion.MC_PlanarMover;
	_ObjectInfo : Tc3_Mc3PlanarMotion.PlanarObjectInfo;
	_std		: CDT_MCTOPLC_PLANAR_MOVER_STD;

	//Command Log
	_CommandLog : ARRAY[0..SystemParameters.MAX_LOG_COUNT] OF ST_CommandLog;

	//Mover Task Declarations
	EnableMover						: FB_Enable(THIS^, Name := 'Enable');
	DisableMover					: FB_Disable(THIS^, Name := 'Disable');
	HaltMover						: FB_Halt(THIS^, Name := 'Halt');
	JoinMoverToTrack				: FB_JoinTrack(THIS^, Name := 'JoinTrack');
	JoinToClosestTrack				: FB_JoinClosestTrack(THIS^, Name := 'JoinClosestTrack');
	LeaveMoverFromTrack				: FB_LeaveTrack(THIS^, Name := 'LeaveTrack');
	ResetMover						: FB_ResetMover(THIS^, Name := 'Reset');
	MoveOnTrackXY					: FB_TrackMoveXY(THIS^, Name := 'MoveOnTrack');
	MoveOnTrack						: FB_TrackMove(THIS^, Name := 'MoveOnTrack');
	RotateMover						: FB_Rotate(THIS^, Name := 'Rotate');
	XMove							: FB_MoveX(THIS^, Name := 'MoveX');
	YMove							: FB_MoveY(THIS^, Name := 'MoveY');
	ZMove							: FB_MoveZ(THIS^, Name := 'MoveZ');
	AMove							: FB_MoveA(THIS^, Name := 'MoveA');
	BMove							: FB_MoveB(THIS^, Name := 'MoveB');
	MoveToPosition					: FB_MoveToPosition(THIS^, Name := 'MoveToPosition');
	XMoveRelative					: FB_MoveRelativeX(THIS^, Name := 'MoveRelativeX');
	YMoveRelative					: FB_MoveRelativeY(THIS^, Name := 'MoveRelativeY');
	CMoveRelative					: FB_MoveRelativeC(THIS^, Name := 'MoveRelativeC');
	XMoveVelocity					: FB_MoveVelocityX(THIS^, Name := 'MoveVelocityX');
	YMoveVelocity					: FB_MoveVelocityY(THIS^, Name := 'MoveVelocityY');
	CMoveVelocity					: FB_MoveVelocityC(THIS^, Name := 'MoveVelocityC');
	AddMoverToGroup					: FB_AddToGroup(THIS^, Name := 'AddToGroup');
	SquareMover						: FB_SquareUp(THIS^, Name := 'SquareUp');
	RunExternalSetpointRelativeMode : FB_RunExternalSetpointRelativeMode(THIS^, Name := 'Run external setpoint relative mode');
	RunExternalSetpointAbsoluteMode : FB_RunExternalSetpointAbsoluteMode(THIS^, Name := 'Run external setpoint absolute mode');
	StopExternalSetpoint			: FB_StopExternalSetpoint(THIS^, Name := 'Stop external setpoint');
	EnterMvmtAreaTask				: FB_EnterMovementArea(THIS^, Name := 'EnterMovementArea');
	LeaveMvmtAreaTask				: FB_LeaveMovementArea(THIS^, Name := 'LeaveMovementArea');
	InvalidCommandResult			: FB_TaskResult := (Busy := FALSE, Error := TRUE, ErrorID := 9999);

	//Internal Vars
	_Initialized		 : BOOL;
	_Busy				 : BOOL;
	_Error				 : BOOL;
	_ErrorID			 : UDINT;
	_MoveDynamics		 : ST_MoveDynamics;
	_RotateDynamics		 : ST_MoveDynamics;
	_TiltDynamics		 : ST_MoveDynamics;
	_DynMove			 : Tc3_Physics.DynamicConstraint_PathXYZ;
	_DynRotate			 : Tc3_Physics.DynamicConstraint_Coordinates;
	_DynTrackMove		 : Tc3_Physics.DynamicConstraint_PathXY;
	_DynHalt			 : Tc3_Physics.DynamicConstraint_Coordinates;
	_Gap				 : LREAL;
	_MoverIndex			 : UDINT;
	_TrackId			 : UDINT;
	_MoverBTN			 : STRING;
	_IdentifiedBTN		 : STRING;
	_MoverType			 : XPlanarMoverType;
	_InStation			 : BOOL;
	_MoverActPos		 : MoverVector;
	_PreviousActPos		 : MoverVector;
	_ClosestQuarterAngle : LREAL;
	_AtRotationPosition	 : BOOL;
	_ModuloPosC			 : LREAL;
	ipDestination		 : I_XPlanarStation;
	ipMoverTcIo			 : I_TcIoXPlanarMover;
	TypeIsRead			 : BOOL;
	UpdateMoveDynamics	 : BOOL;
	UpdateRotateDynamics : BOOL;
	UpdateTiltDynamics	 : BOOL;
	ClosestSquarePos	 : LREAL;
	ToMCMapStatus		 : EPlcMappingStatus;
	FromMCMapStatus		 : EPlcMappingStatus;
	LinkErrMsg			 : BOOL;
	_MoverData			 : I_MoverData := NullObjects.MoverData;
END_VAR

METHOD Initialize
//Set initial dynamics

//Halt
_DynHalt.SetLimit(Coord_Mcs_X,
				  500.0,
				  10000.0,
				  10000.0,
				  100000.0);

_DynHalt.SetLimit(Coord_Mcs_Y,
				  500.0,
				  10000.0,
				  10000.0,
				  100000.0);

_DynHalt.SetLimit(Coord_Mcs_Z,
				  500.0,
				  10000.0,
				  10000.0,
				  100000.0);

_DynHalt.SetLimit(Coord_Mcs_A1,
				  10.0,
				  100.0,
				  100.0,
				  100.0);

_DynHalt.SetLimit(Coord_Mcs_B1,
				  10.0,
				  100.0,
				  100.0,
				  100.0);

_DynHalt.SetLimit(Coord_Mcs_C1,
				  36.0,
				  360.0,
				  360.0,
				  360.0);

//XY Movement
_DynMove.SetValuesVADJ(200,
					   2000,
					   2000,
					   50000);

_DynTrackMove.SetValuesVADJ(200,
							2000,
							2000,
							50000);

//Rotation
_DynRotate.SetLimit(Coord_Mcs_A1,
					100,
					5000,
					5000,
					50000);

_DynRotate.SetLimit(Coord_Mcs_B1,
					100,
					5000,
					5000,
					50000);

_DynRotate.SetLimit(Coord_Mcs_C1,
					100,
					5000,
					5000,
					50000);

//Safe Gap Value
_Gap := 200;


//Make sure mover is linkted to MC3 Object
_ObjectInfo := _Mover.GetPlanarObjectInfo();
IF _ObjectInfo.Id = 0 THEN
	IF NOT LinkErrMsg THEN
		ADSLOGDINT(ADSLOG_MSGTYPE_ERROR, 'Object not linked to MC! Mover: %d', TO_DINT(_MoverIndex));
		LinkErrMsg := TRUE;
	END_IF
	RETURN;
END_IF

//Get mover info and load mover object data
IF ipMoverTcIo <> 0 THEN
	_MoverBTN  := ipMoverTcIo.GetBtn();
	_MoverType := ipMoverTcIo.GetMoverType();
	IF _MoverIndex > 0 AND _MoverIndex <= HmiObjectCounts.Movers THEN
		CASE _MoverType OF
			XPlanarMoverType.APM4220:
				XPlanarHMI.MoverObjects[_MoverIndex].Width	:= 115;
				XPlanarHMI.MoverObjects[_MoverIndex].Height := 115;

			XPlanarMoverType.APM4221:
				XPlanarHMI.MoverObjects[_MoverIndex].Width	:= 127;
				XPlanarHMI.MoverObjects[_MoverIndex].Height := 127;

			XPlanarMoverType.APM4230:
				XPlanarHMI.MoverObjects[_MoverIndex].Width	:= 115;
				XPlanarHMI.MoverObjects[_MoverIndex].Height := 155;

			XPlanarMoverType.APM4330:
				XPlanarHMI.MoverObjects[_MoverIndex].Width	:= 155;
				XPlanarHMI.MoverObjects[_MoverIndex].Height := 155;

			XPlanarMoverType.APM4330_0001:
				XPlanarHMI.MoverObjects[_MoverIndex].Width	:= 150;
				XPlanarHMI.MoverObjects[_MoverIndex].Height := 150;

			XPlanarMoverType.APM4350:
				XPlanarHMI.MoverObjects[_MoverIndex].Width	:= 155;
				XPlanarHMI.MoverObjects[_MoverIndex].Height := 235;

			XPlanarMoverType.APM4550:
				XPlanarHMI.MoverObjects[_MoverIndex].Width	:= 235;
				XPlanarHMI.MoverObjects[_MoverIndex].Height := 235;
		END_CASE
	END_IF
	
	_Initialized := TRUE;
END_IF
END_METHOD

{attribute 'monitoring' := 'call'}
PROPERTY Initialized : BOOL
GET
Initialized := _Initialized;
END_GET
SET
_Initialized := Initialized;
END_SET
END_PROPERTY

METHOD FreeMove : I_PlanarTaskResult
VAR_INPUT
	XTarget			: LREAL;
	YTarget			: LREAL;
	CTarget			: LREAL := 0;
	Rototranslation : BOOL	:= FALSE;
END_VAR
FreeMove := MoveToPosition.Execute(XTarget, YTarget, CTarget, _DynMove, Rototranslation);
END_METHOD

METHOD JoinClosestTrack : I_PlanarTaskResult
VAR_INPUT
	UseOrientation : BOOL := FALSE;
END_VAR
JoinClosestTrack := JoinToClosestTrack.Execute(UseOrientation, _DynMove);
END_METHOD

METHOD JoinTrack : I_PlanarTaskResult
VAR_INPUT
	ipTrack		   : I_XPlanarTrack;
	UseOrientation : BOOL := FALSE;
END_VAR
JoinTrack := JoinMoverToTrack.Execute(ipTrack, UseOrientation, _DynMove);
END_METHOD

METHOD LeaveTrack : I_PlanarTaskResult
VAR_INPUT
	DestinationX   : LREAL;
	DestinationY   : LREAL;
	UseOrientation : BOOL := FALSE;
END_VAR

VAR_INST
	Destination : PositionXYC;
END_VAR
LeaveTrack := LeaveMoverFromTrack.Execute(DestinationX,
										  DestinationY,
										  UseOrientation,
										  _DynMove);
END_METHOD

METHOD MoveRelativeC : I_PlanarTaskResult
VAR_INPUT
	Distance	: LREAL;
END_VAR
MoveRelativeC := CMoveRelative.Execute(Distance, _DynRotate);
END_METHOD

METHOD MoveRelativeX : I_PlanarTaskResult
VAR_INPUT
	Distance	: LREAL;
END_VAR
MoveRelativeX := XMoveRelative.Execute(Distance, _DynMove);
END_METHOD

METHOD MoveRelativeY : I_PlanarTaskResult
VAR_INPUT
	Distance	: LREAL;
END_VAR
MoveRelativeY := YMoveRelative.Execute(Distance, _DynMove);
END_METHOD

METHOD MoveVelocityC : I_PlanarTaskResult
VAR_INPUT
	Velocity	: LREAL;
END_VAR
MoveVelocityC := CMoveVelocity.Execute(Velocity, _DynRotate);
END_METHOD

METHOD MoveVelocityX : I_PlanarTaskResult
VAR_INPUT
	Velocity	: LREAL;
END_VAR
MoveVelocityX := XMoveVelocity.Execute(Velocity, _DynMove);
END_METHOD

METHOD MoveVelocityY : I_PlanarTaskResult
VAR_INPUT
	Velocity	: LREAL;
END_VAR
MoveVelocityY := YMoveVelocity.Execute(Velocity, _DynMove);
END_METHOD

METHOD MoveX : I_PlanarTaskResult
VAR_INPUT
	Position	: LREAL;
END_VAR
MoveX := XMove.Execute(Position, _DynMove);
END_METHOD

METHOD MoveY : I_PlanarTaskResult
VAR_INPUT
	Position	: LREAL;
END_VAR
MoveY := YMove.Execute(Position, _DynMove);
END_METHOD

METHOD Rotate : I_PlanarTaskResult
VAR_INPUT
	Position		: LREAL;
	AdditionalTurns : DINT := 0;
END_VAR

VAR
	Direction : Tc3_Mc3PlanarMotion.MC_DIRECTION;
END_VAR
IF AdditionalTurns < 0 OR Position < 0 THEN
	Direction := Tc3_Mc3PlanarMotion.MC_DIRECTION.mcDirectionNegative;
ELSIF Position = 0 AND AdditionalTurns = 0 THEN
	Direction := Tc3_Mc3PlanarMotion.MC_DIRECTION.mcDirectionShortestWay;
ELSE
	Direction := Tc3_Mc3PlanarMotion.MC_DIRECTION.mcDirectionPositive;
END_IF

IF _AtRotationPosition OR ((Position >= -10 OR Position <= 10) AND AdditionalTurns = 0) THEN
	Rotate := RotateMover.Execute(ABS(Position),
								  ABS(AdditionalTurns),
								  Direction,
								  _DynRotate);
ELSE
	Rotate := InvalidCommandResult;
END_IF
END_METHOD

METHOD RunExternalSpAbsoluteMode : I_PlanarTaskResult
VAR_INPUT
	Position	 : MoverVector;
	Velocity	 : MoverVector;
	Acceleration : MoverVector;
END_VAR
RunExternalSpAbsoluteMode := RunExternalSetpointAbsoluteMode.Execute(Position,Velocity,Acceleration);
END_METHOD

METHOD RunExternalSpRelativeMode : I_PlanarTaskResult
VAR_INPUT
	Position	 : MoverVector;
	Velocity	 : MoverVector;
	Acceleration : MoverVector;
END_VAR
RunExternalSpRelativeMode := RunExternalSetpointRelativeMode.Execute(Position,Velocity,Acceleration);
END_METHOD

METHOD SendToStation : I_PlanarTaskResult
VAR_INPUT
	Destination : I_XPlanarStation;
END_VAR

VAR_INST
	CorrectedPos : PositionXYC;
	OnTrackPos	 : LREAL;
END_VAR
ipDestination := Destination; //Update the destination field of the mover
IF _Mover.MCTOPLC.STD.CommandMode = MC_PLANAR_MOVER_COMMAND_MODE.OnTrack THEN
	IF Destination.TrackID <> 0 THEN
		SendToStation := MoveOnTrackXY.Execute(Destination.Position.x,
											   Destination.Position.y,
											   _Gap,
											   ip.Tracks[Destination.TrackID],
											   _DynTrackMove,
											   Tc3_Mc3PlanarMotion.MC_DIRECTION.mcDirectionPositive);
	ELSE
		SendToStation := InvalidCommandResult;
	END_IF
ELSIF _Mover.MCTOPLC.STD.CommandMode = MC_PLANAR_MOVER_COMMAND_MODE.FreeMovement THEN
	CorrectedPos.SetValuesXYC(Destination.Position.x, Destination.Position.y, _MoverActPos.c);
	SendToStation := MoveToPosition.Execute(Destination.Position.x, Destination.Position.y, Destination.Position.c,  _DynMove);
ELSE
	SendToStation := InvalidCommandResult;
END_IF
END_METHOD

METHOD SquareUp : I_PlanarTaskResult
SquareUp := SquareMover.Execute(_ClosestQuarterAngle, _DynRotate, _DynMove);
END_METHOD

METHOD StopExternalSp : I_PlanarTaskResult
StopExternalSp := StopExternalSetpoint.Execute();
END_METHOD

METHOD TiltA : I_PlanarTaskResult
VAR_INPUT
	Position : LREAL;
END_VAR
TiltA := AMove.Execute(Position, _DynRotate);
END_METHOD

METHOD TiltB : I_PlanarTaskResult
VAR_INPUT
	Position : LREAL;
END_VAR
TiltB := BMove.Execute(Position, _DynRotate);
END_METHOD

METHOD TrackMove : I_PlanarTaskResult
VAR_INPUT
	Position : LREAL;
	Gap		  : LREAL;
	Track	  : I_XPlanarTrack;
	Direction : Tc3_Mc3PlanarMotion.MC_DIRECTION;
END_VAR

VAR
	WorkingGap : LREAL;
END_VAR
IF Gap > 0 THEN
	WorkingGap := Gap;
ELSE
	WorkingGap := _Gap;
END_IF

IF Track <> 0 THEN
	TrackMove := MoveOnTrack.Execute(Position,
									 WorkingGap,
									 Track,
									 _DynTrackMove,
									 Direction);
ELSE
	TrackMove := InvalidCommandResult;
END_IF
END_METHOD

METHOD TrackMoveXY : I_PlanarTaskResult
VAR_INPUT
	XPosition : LREAL;
	YPosition : LREAL;
	Gap		  : LREAL;
	Track	  : I_XPlanarTrack;
	Direction : Tc3_Mc3PlanarMotion.MC_DIRECTION;
END_VAR

VAR
	WorkingGap : LREAL;
END_VAR

VAR_INST
	Position   : PositionXYC;
	OnTrackPos : LREAL;
END_VAR
IF Gap > 0 THEN
	WorkingGap := Gap;
ELSE
	WorkingGap := _Gap;
END_IF

IF Track <> 0 THEN
	TrackMoveXY := MoveOnTrackXY.Execute(XPosition,
										 YPosition,
										 WorkingGap,
										 Track,
										 _DynTrackMove,
										 Direction);
ELSE
	TrackMoveXY := InvalidCommandResult;
END_IF
END_METHOD

METHOD VerticalMove : I_PlanarTaskResult
VAR_INPUT
	Position : LREAL;
END_VAR
VerticalMove := ZMove.Execute(Position, _DynMove);
END_METHOD

{attribute 'suppress_wrn_C0410'}
PROPERTY Movement : REFERENCE TO ST_MoveDynamics
GET
Movement REF= _MoveDynamics;
UpdateMoveDynamics := TRUE;
END_GET
END_PROPERTY

{attribute 'suppress_wrn_C0410'}
PROPERTY Rotation : REFERENCE TO ST_MoveDynamics
GET
Rotation REF= _RotateDynamics;
UpdateRotateDynamics := true;
END_GET
END_PROPERTY

{attribute 'suppress_wrn_C0410'}
PROPERTY Tilt : REFERENCE TO ST_MoveDynamics
GET
Tilt REF= _TiltDynamics;
UpdateTiltDynamics := TRUE;
END_GET
END_PROPERTY

{attribute 'suppress_wrn_C0410'}
PROPERTY ActualPosition : REFERENCE TO MoverVector
GET
ActualPosition ref= _MoverActPos;
END_GET
END_PROPERTY

//Adds the mover object to the overall XPlanar CA group
METHOD AddToGroup : I_PlanarTaskResult
VAR_INPUT
	PlanarGroup : REFERENCE TO MC_PlanarGroup;
END_VAR
AddToGroup := AddMoverToGroup.Execute(PlanarGroup);
END_METHOD

PROPERTY AtRotationPosition : BOOL
GET
AtRotationPosition := _AtRotationPosition;
END_GET
END_PROPERTY

PROPERTY Busy : BOOL
GET
Busy := _Busy;
END_GET
END_PROPERTY

{attribute 'suppress_wrn_C0410'}
PROPERTY CommandLog : REFERENCE TO ARRAY [0..SystemParameters.MAX_LOG_COUNT] of ST_CommandLog
GET
CommandLog ref= _CommandLog;
END_GET
END_PROPERTY

PROPERTY Destination : I_XPlanarStation
GET
Destination := ipDestination;
END_GET
SET
ipDestination := Destination;
END_SET
END_PROPERTY

METHOD Disable : I_PlanarTaskResult
Disable := DisableMover.Execute();
END_METHOD

PROPERTY Dynamics : I_MoveDynamics
GET
Dynamics := THIS^;
END_GET
END_PROPERTY

METHOD Enable : I_PlanarTaskResult
Enable := EnableMover.Execute();
END_METHOD

METHOD EnterMovementArea : I_PlanarTaskResult
VAR_INPUT
	PartId		: OTCID;
	PositionX	: LREAL;
	PositionY	: LREAL;
END_VAR
IF PartID = 0 AND PositionX < 0 OR PositionY < 0 THEN
	EnterMovementArea := InvalidCommandResult;
ELSE
	EnterMovementArea := EnterMvmtAreaTask.Execute(PartId, PositionX, PositionY);
END_IF
END_METHOD

PROPERTY Error : BOOL
GET
Error := _Error;
END_GET
END_PROPERTY

PROPERTY ErrorId : UDINT
GET
ErrorId := ErrorID;
END_GET
END_PROPERTY

PROPERTY Gap : LREAL
GET
Gap := _Gap;
END_GET
SET
_Gap := Gap;
END_SET
END_PROPERTY

METHOD Halt : I_PlanarTaskResult
Halt := HaltMover.Execute(_DynHalt);
END_METHOD

